(* IEC 61131-3 sources: SmartHomeNew/ (part 9) *)

(* ---- FB_System_Scenario_Arbitration.st ---- *)
// ==============================================================================
// System scenario arbitration helper
//
// Internal helper for PRG_System.
// Owns scenario request validation, priority resolution, fail-safe clamp,
// degraded-mode adaptation, policy logging, and FB_Scenario_Manager call.
// ==============================================================================
FUNCTION_BLOCK FB_System_Scenario_Arbitration
VAR_INPUT
    VI_System_Time_MS : UDINT;
    VI_IsActivePLC : BOOL;
    VI_System_Mode : E_System_Operating_Mode;
    VI_Security_Armed : BOOL;
END_VAR

VAR_IN_OUT
    VIO_Scenario_Req_Operator : E_SCENARIO_TYPE;
    VIO_Scenario_Req_Gateway : E_SCENARIO_TYPE;
    VIO_Scenario_Req_Rule : E_SCENARIO_TYPE;
    VIO_Scenario_Req_Final : E_SCENARIO_TYPE;
    VIO_Scenario_Intent : E_SCENARIO_TYPE;
    VIO_Scenario_Source : E_SCENARIO_SOURCE;
END_VAR

VAR
    fbLogEvent : FB_LogEvent;
    fbScenarioManager : FB_Scenario_Manager;
    L_Restore_Target : E_SCENARIO_TYPE;
END_VAR

// === SCENARIO REQUEST VALIDATION ===
// Normalize invalid values to NONE to avoid corrupt inputs.
// Actual enum range in E_SCENARIO_TYPE is 0..7.
IF TO_USINT(VIO_Scenario_Req_Operator) > 7 THEN
    VIO_Scenario_Req_Operator := E_SCENARIO_TYPE.SCENARIO_NONE;
END_IF;

IF TO_USINT(VIO_Scenario_Req_Gateway) > 7 THEN
    VIO_Scenario_Req_Gateway := E_SCENARIO_TYPE.SCENARIO_NONE;
END_IF;

IF TO_USINT(VIO_Scenario_Req_Rule) > 7 THEN
    VIO_Scenario_Req_Rule := E_SCENARIO_TYPE.SCENARIO_NONE;
END_IF;

// === SCENARIO PRIORITY RESOLUTION ===
// Produces VIO_Scenario_Req_Final (TRACE ONLY, not executed directly)
IF VI_System_Mode = E_System_Operating_Mode.MODE_SAFE_STOP THEN
    VIO_Scenario_Req_Final := 0;
    VIO_Scenario_Source := SRC_SAFETY;
ELSIF VIO_Scenario_Req_Operator <> 0 THEN
    VIO_Scenario_Req_Final := VIO_Scenario_Req_Operator;
    VIO_Scenario_Source := SRC_OPERATOR;
ELSIF VIO_Scenario_Req_Gateway <> 0 THEN
    VIO_Scenario_Req_Final := VIO_Scenario_Req_Gateway;
    VIO_Scenario_Source := SRC_GATEWAY;
ELSIF VIO_Scenario_Req_Rule <> 0 THEN
    VIO_Scenario_Req_Final := VIO_Scenario_Req_Rule;
    VIO_Scenario_Source := SRC_RULE;
ELSE
    VIO_Scenario_Req_Final := GVL_STATUS.G_Current_Scenario;
    VIO_Scenario_Source := SRC_NONE;
END_IF;

VIO_Scenario_Intent := VIO_Scenario_Req_Final;

// === FAIL-SAFE SCENARIO CLAMP ===
CASE VI_System_Mode OF
    E_System_Operating_Mode.MODE_SAFE_STOP:
        VIO_Scenario_Intent := E_SCENARIO_TYPE.SCENARIO_NONE;

    E_System_Operating_Mode.MODE_FREEZE_PROTECTION:
        VIO_Scenario_Intent := E_SCENARIO_TYPE.SCENARIO_NONE;

    E_System_Operating_Mode.MODE_DEGRADED:
        CASE VIO_Scenario_Intent OF
            E_SCENARIO_TYPE.SCENARIO_NONE,
            E_SCENARIO_TYPE.SCENARIO_PRESENCE,
            E_SCENARIO_TYPE.SCENARIO_AWAY,
            E_SCENARIO_TYPE.SCENARIO_SLEEP:
                ; // allowed in degraded
        ELSE
            VIO_Scenario_Intent := E_SCENARIO_TYPE.SCENARIO_NONE;
        END_CASE;
END_CASE;

// === CONTEXT FAIL-SAFE AUTOMATION ===
// If security is armed and no explicit source is requesting another scenario,
// force safe occupancy context to AWAY while system remains in MODE_NORMAL.
IF VI_System_Mode = E_System_Operating_Mode.MODE_NORMAL THEN
    IF VI_Security_Armed AND
       (VIO_Scenario_Req_Operator = E_SCENARIO_TYPE.SCENARIO_NONE) AND
       (VIO_Scenario_Req_Gateway = E_SCENARIO_TYPE.SCENARIO_NONE) AND
       (VIO_Scenario_Req_Rule = E_SCENARIO_TYPE.SCENARIO_NONE) AND
       (VIO_Scenario_Intent <> E_SCENARIO_TYPE.SCENARIO_AWAY) THEN

        IF (VIO_Scenario_Intent <> E_SCENARIO_TYPE.SCENARIO_NONE) AND
           (VIO_Scenario_Intent <> E_SCENARIO_TYPE.SCENARIO_AWAY) THEN
            GVL_POLICY.G_Away_Previous_Scenario := VIO_Scenario_Intent;
        ELSIF (GVL_STATUS.G_Current_Scenario <> E_SCENARIO_TYPE.SCENARIO_NONE) AND
              (GVL_STATUS.G_Current_Scenario <> E_SCENARIO_TYPE.SCENARIO_AWAY) THEN
            GVL_POLICY.G_Away_Previous_Scenario := GVL_STATUS.G_Current_Scenario;
        ELSE
            GVL_POLICY.G_Away_Previous_Scenario := E_SCENARIO_TYPE.SCENARIO_PRESENCE;
        END_IF;

        VIO_Scenario_Intent := E_SCENARIO_TYPE.SCENARIO_AWAY;
        VIO_Scenario_Source := SRC_POLICY;

        fbLogEvent(
            VI_Event_Type := 5,
            VI_Timestamp := VI_System_Time_MS,
            VI_Param1 := TO_UDINT(VIO_Scenario_Source),
            VI_Param2 := TO_UDINT(E_SCENARIO_TYPE.SCENARIO_AWAY)
        );
    END_IF;

    // When security is disarmed and no explicit source requests AWAY,
    // leave AWAY and return to the scenario captured before short-away arming.
    IF (NOT VI_Security_Armed) AND
       (VIO_Scenario_Req_Operator = E_SCENARIO_TYPE.SCENARIO_NONE) AND
       (VIO_Scenario_Req_Gateway = E_SCENARIO_TYPE.SCENARIO_NONE) AND
       (VIO_Scenario_Req_Rule = E_SCENARIO_TYPE.SCENARIO_NONE) AND
       (VIO_Scenario_Intent = E_SCENARIO_TYPE.SCENARIO_AWAY) AND
       GVL_POLICY.G_Away_Active THEN

        L_Restore_Target := GVL_POLICY.G_Away_Previous_Scenario;

        IF (L_Restore_Target = E_SCENARIO_TYPE.SCENARIO_NONE) OR
           (L_Restore_Target = E_SCENARIO_TYPE.SCENARIO_AWAY) THEN
            L_Restore_Target := E_SCENARIO_TYPE.SCENARIO_PRESENCE;
        END_IF;

        VIO_Scenario_Intent := L_Restore_Target;
        VIO_Scenario_Source := SRC_POLICY;
    END_IF;
END_IF;

// === DEGRADED-AWARE SCENARIO ADAPTATION ===
// Soft adaptation in degraded mode: keep explicit requests intact,
// but if no source is requesting a scenario, move behavior to a safer baseline.
IF VI_System_Mode = E_System_Operating_Mode.MODE_DEGRADED THEN
    IF (VIO_Scenario_Req_Operator = E_SCENARIO_TYPE.SCENARIO_NONE) AND
       (VIO_Scenario_Req_Gateway = E_SCENARIO_TYPE.SCENARIO_NONE) AND
       (VIO_Scenario_Req_Rule = E_SCENARIO_TYPE.SCENARIO_NONE) THEN

        IF VI_Security_Armed THEN
            IF VIO_Scenario_Intent <> E_SCENARIO_TYPE.SCENARIO_AWAY THEN
                IF (VIO_Scenario_Intent <> E_SCENARIO_TYPE.SCENARIO_NONE) AND
                   (VIO_Scenario_Intent <> E_SCENARIO_TYPE.SCENARIO_AWAY) THEN
                    GVL_POLICY.G_Away_Previous_Scenario := VIO_Scenario_Intent;
                ELSE
                    GVL_POLICY.G_Away_Previous_Scenario := E_SCENARIO_TYPE.SCENARIO_PRESENCE;
                END_IF;

                VIO_Scenario_Intent := E_SCENARIO_TYPE.SCENARIO_AWAY;
                VIO_Scenario_Source := SRC_POLICY;

                fbLogEvent(
                    VI_Event_Type := 6,
                    VI_Timestamp := VI_System_Time_MS,
                    VI_Param1 := TO_UDINT(VIO_Scenario_Source),
                    VI_Param2 := TO_UDINT(E_SCENARIO_TYPE.SCENARIO_AWAY)
                );
            END_IF;

        ELSIF VIO_Scenario_Intent = E_SCENARIO_TYPE.SCENARIO_PRESENCE THEN
            IF VIO_Scenario_Intent <> E_SCENARIO_TYPE.SCENARIO_SLEEP THEN
                VIO_Scenario_Intent := E_SCENARIO_TYPE.SCENARIO_SLEEP;
                VIO_Scenario_Source := SRC_POLICY;

                fbLogEvent(
                    VI_Event_Type := 7,
                    VI_Timestamp := VI_System_Time_MS,
                    VI_Param1 := TO_UDINT(VIO_Scenario_Source),
                    VI_Param2 := TO_UDINT(E_SCENARIO_TYPE.SCENARIO_SLEEP)
                );
            END_IF;
        END_IF;
    END_IF;
END_IF;

fbScenarioManager(
    VI_System_Time_MS := VI_System_Time_MS,
    VI_Activate_Request := VIO_Scenario_Intent,
    VI_IsActivePLC := VI_IsActivePLC,
    VI_System_Mode := VI_System_Mode,
    VO_Current_Scenario => GVL_STATUS.G_Current_Scenario
);

// >>> BULK_SYNC_ANCHOR: FB_System_Scenario_Arbitration <<<
END_FUNCTION_BLOCK

(* ---- FB_System_Timebase.st ---- *)
// ==============================================================================
// System timebase helper
//
// Internal helper for PRG_System.
// Owns PLC runtime clock projection into GVL_STATUS:
// - monotonic system milliseconds
// - time-of-day milliseconds
// - day of week / day of year rollover
// - TOD representation
// ==============================================================================
FUNCTION_BLOCK FB_System_Timebase
VAR
    L_Time_Diff : UDINT;
END_VAR

GVL_STATUS.G_System_Time_MS := TIME_TO_UDINT(TIME());

L_Time_Diff := SEL(
    GVL_STATUS.G_System_Time_MS >= GVL_STATUS.G_Last_System_Time_MS,
    GVL_STATUS.G_System_Time_MS - GVL_STATUS.G_Last_System_Time_MS,
    (4294967295 - GVL_STATUS.G_Last_System_Time_MS) + GVL_STATUS.G_System_Time_MS + 1
);

GVL_STATUS.G_Time_Of_Day_MS := (GVL_STATUS.G_Time_Of_Day_MS + L_Time_Diff) MOD 86400000;

IF GVL_STATUS.G_Time_Of_Day_MS < L_Time_Diff THEN
    GVL_STATUS.G_Current_Day := (GVL_STATUS.G_Current_Day MOD 7) + 1;
    GVL_STATUS.G_Day_Of_Year := (GVL_STATUS.G_Day_Of_Year MOD 365) + 1;
END_IF;

GVL_STATUS.G_Last_System_Time_MS := GVL_STATUS.G_System_Time_MS;
GVL_STATUS.G_Current_TOD := UDINT_TO_TOD(GVL_STATUS.G_Time_Of_Day_MS);

// >>> BULK_SYNC_ANCHOR: FB_System_Timebase <<<
END_FUNCTION_BLOCK

(* ---- FB_Time_Service.st ---- *)
FUNCTION_BLOCK FB_Time_Service
VAR
    L_Real_Now : UDINT;
    L_Elapsed : UDINT;
    L_Scaled_Delta : UDINT;
END_VAR

// read real time
L_Real_Now := GVL_STATUS.G_System_Time_MS;

// wrap-safe delta (real time base)
IF L_Real_Now >= GVL_TIME_SERVICE.G_Last_Now_MS THEN
    L_Elapsed := L_Real_Now - GVL_TIME_SERVICE.G_Last_Now_MS;
    GVL_TIME_SERVICE.G_Wrap_Detected := FALSE;
ELSE
    L_Elapsed := (16#FFFFFFFF - GVL_TIME_SERVICE.G_Last_Now_MS) + L_Real_Now + 1;
    GVL_TIME_SERVICE.G_Wrap_Detected := TRUE;
END_IF;

GVL_TIME_SERVICE.G_Last_Now_MS := L_Real_Now;

// --- SIMULATION MODE ---
IF GVL_TIME_SERVICE.G_Sim_Enabled THEN

    IF NOT GVL_TIME_SERVICE.G_Sim_Frozen THEN
        // scale delta
        L_Scaled_Delta := UDINT(REAL(L_Elapsed) * GVL_TIME_SERVICE.G_Sim_Time_Scale);

        // advance simulated absolute time
        GVL_TIME_SERVICE.G_Sim_Now_MS := GVL_TIME_SERVICE.G_Sim_Now_MS + L_Scaled_Delta;

        // advance TOD with wrap
        GVL_TIME_SERVICE.G_Sim_Time_Of_Day_MS := GVL_TIME_SERVICE.G_Sim_Time_Of_Day_MS + L_Scaled_Delta;

        IF GVL_TIME_SERVICE.G_Sim_Time_Of_Day_MS >= 86400000 THEN
            GVL_TIME_SERVICE.G_Sim_Time_Of_Day_MS := GVL_TIME_SERVICE.G_Sim_Time_Of_Day_MS MOD 86400000;
            GVL_TIME_SERVICE.G_Sim_Day_Of_Week := GVL_TIME_SERVICE.G_Sim_Day_Of_Week + 1;
            IF GVL_TIME_SERVICE.G_Sim_Day_Of_Week > 7 THEN
                GVL_TIME_SERVICE.G_Sim_Day_Of_Week := 1;
            END_IF;
        END_IF;
    END_IF;

    // publish simulated time
    GVL_TIME_SERVICE.G_Now_MS := GVL_TIME_SERVICE.G_Sim_Now_MS;
    GVL_TIME_SERVICE.G_Time_Of_Day_MS := GVL_TIME_SERVICE.G_Sim_Time_Of_Day_MS;
    GVL_TIME_SERVICE.G_Day_Of_Week := GVL_TIME_SERVICE.G_Sim_Day_Of_Week;

ELSE
    // publish real time
    GVL_TIME_SERVICE.G_Now_MS := L_Real_Now;
    GVL_TIME_SERVICE.G_Time_Of_Day_MS := GVL_STATUS.G_Time_Of_Day_MS;
    GVL_TIME_SERVICE.G_Day_Of_Week := INT(GVL_STATUS.G_Current_Day);
END_IF;

// publish delta (always based on real time)
GVL_TIME_SERVICE.G_Delta_MS := L_Elapsed;

END_FUNCTION_BLOCK

(* ---- FB_Trace_Logger.st ---- *)
FUNCTION_BLOCK FB_Trace_Logger
VAR_INPUT
    VI_Event_Code : INT;
    VI_System_Time : UDINT;
END_VAR

GVL_TRACE.G_Trace_Index := GVL_TRACE.G_Trace_Index + 1;
IF GVL_TRACE.G_Trace_Index > GVL_TRACE.G_Trace_Max THEN
    GVL_TRACE.G_Trace_Index := 1;
END_IF;

GVL_TRACE.G_Trace_Time[GVL_TRACE.G_Trace_Index] := VI_System_Time;
GVL_TRACE.G_Trace_Code[GVL_TRACE.G_Trace_Index] := VI_Event_Code;
END_FUNCTION_BLOCK

(* ---- FB_Trace_Write.st ---- *)
FUNCTION_BLOCK FB_Trace_Write
VAR_INPUT
    iLayer : E_Trace_Layer;
    iSource : E_Trace_Source;
    iReason : E_System_Reason_Code;
    iValueBool : BOOL;
    iValueReal : REAL;
    iText : STRING(120);
END_VAR

VAR
    L_Index : INT;
END_VAR

IF NOT GVL_TRACE.G_Trace_Enabled THEN RETURN; END_IF;

L_Index := GVL_TRACE.G_Trace_Write_Index;

GVL_TRACE.G_Trace_Buffer[L_Index].Timestamp_MS := GVL_TIME_SERVICE.G_Now_MS;
GVL_TRACE.G_Trace_Buffer[L_Index].Layer := iLayer;
GVL_TRACE.G_Trace_Buffer[L_Index].Source := iSource;
GVL_TRACE.G_Trace_Buffer[L_Index].Reason_Code := iReason;
GVL_TRACE.G_Trace_Buffer[L_Index].Value_Bool := iValueBool;
GVL_TRACE.G_Trace_Buffer[L_Index].Value_Real := iValueReal;
GVL_TRACE.G_Trace_Buffer[L_Index].Text := iText;

L_Index := L_Index + 1;
IF L_Index > 200 THEN L_Index := 1; END_IF;

GVL_TRACE.G_Trace_Write_Index := L_Index;

(* ---- FB_Trend_Analyzer.st ---- *)
FUNCTION_BLOCK FB_Trend_Analyzer
VAR_INPUT
    VI_Count      : INT;
END_VAR
VAR_IN_OUT
    VI_Data       : ARRAY[1..GVL_CONSTANTS.C_MAX_TREND_DATA_POINTS] OF REAL;
END_VAR
VAR_OUTPUT
    VO_Average    : REAL;
    VO_Max        : REAL;
    VO_Min        : REAL;
    VO_Trend_Up   : BOOL;
    VO_Trend_Down : BOOL;
END_VAR
VAR
    L_i   : INT;
    L_Sum : REAL;
END_VAR

VO_Average := 0.0;
VO_Max := 0.0;
VO_Min := 0.0;
VO_Trend_Up := FALSE;
VO_Trend_Down := FALSE;

IF VI_Count > 0 AND VI_Count <= GVL_CONSTANTS.C_MAX_TREND_DATA_POINTS THEN
    VO_Max := VI_Data[1];
    VO_Min := VI_Data[1];
    L_Sum := 0.0;

    FOR L_i := 1 TO VI_Count DO
        IF VI_Data[L_i] > VO_Max THEN VO_Max := VI_Data[L_i]; END_IF;
        IF VI_Data[L_i] < VO_Min THEN VO_Min := VI_Data[L_i]; END_IF;
        L_Sum := L_Sum + VI_Data[L_i];
    END_FOR;

    VO_Average := L_Sum / INT_TO_REAL(VI_Count);

    IF VI_Count >= 2 THEN
        VO_Trend_Up := (VI_Data[VI_Count] > VI_Data[1]);
        VO_Trend_Down := (VI_Data[VI_Count] < VI_Data[1]);
    END_IF;
END_IF;
END_FUNCTION_BLOCK

(* ---- FB_Trend_Logger.st ---- *)
FUNCTION_BLOCK FB_Trend_Logger
VAR_INPUT
    VI_System_Time_MS : UDINT;
    VI_Config : ST_Trend_Config;
    VI_Current_Value : REAL;
END_VAR
VAR_OUTPUT
    VO_Data : ST_Trend_Data;
END_VAR
VAR
    L_Last_Log_Time : UDINT;
    L_Last_Value : REAL;
    L_Deviation : REAL;
    L_Elapsed_Time : UDINT;
    L_Write_Index : UDINT;
END_VAR

IF NOT VI_Config.enabled THEN
    RETURN;
END_IF;

L_Deviation := ABS(VI_Current_Value - L_Last_Value);
L_Elapsed_Time := SEL(
    VI_System_Time_MS >= L_Last_Log_Time,
    VI_System_Time_MS - L_Last_Log_Time,
    (4294967295 - L_Last_Log_Time) + VI_System_Time_MS + 1
);

IF (L_Deviation >= (ABS(L_Last_Value) * VI_Config.deviation_threshold_percent / REAL#100.0)) OR
   (L_Elapsed_Time >= GVL_CONSTANTS.C_MS_IN_HOUR) THEN

    L_Write_Index := (VO_Data.record_count MOD 100) + 1;
    VO_Data.write_index := L_Write_Index;
    VO_Data.values[L_Write_Index] := VI_Current_Value;
    VO_Data.timestamps[L_Write_Index] := VI_System_Time_MS;
    VO_Data.record_count := VO_Data.record_count + 1;
    VO_Data.sum_values := VO_Data.sum_values + VI_Current_Value;
    VO_Data.config := VI_Config;

    L_Last_Value := VI_Current_Value;
    L_Last_Log_Time := VI_System_Time_MS;
END_IF;

END_FUNCTION_BLOCK

(* ---- FB_Valve_Test_Manager.st ---- *)
FUNCTION_BLOCK FB_Valve_Test_Manager
VAR_INPUT
    VI_System_Time_MS : UDINT;
    VI_IsActivePLC : BOOL;
END_VAR
VAR_IN_OUT
    VI_Valve_Currents : ARRAY[1..GVL_CONSTANTS.C_MAX_MANIFOLDS] OF REAL;
    VI_Valve_End_Switches : ARRAY[1..GVL_CONSTANTS.C_MAX_MANIFOLDS] OF BOOL;
    VI_Config : ARRAY[1..GVL_CONSTANTS.C_MAX_MANIFOLDS] OF ST_Valve_Test_Config;
END_VAR
VAR_OUTPUT
    VO_Test_Active : BOOL;
    VO_Current_Valve : INT; // Текущий тестируемый клапан
    VO_Valve_Cmd : ARRAY[1..GVL_CONSTANTS.C_MAX_MANIFOLDS] OF BOOL;
    VO_Test_Results : ARRAY[1..GVL_CONSTANTS.C_MAX_MANIFOLDS] OF BOOL; // TRUE = OK
    VO_Status_Msg : STRING(200);
END_VAR
VAR
    L_State : INT;
    L_Current_Valve : INT := 1;
    L_Test_Start_Time : UDINT;
    L_Last_Test_Time : ARRAY[1..GVL_CONSTANTS.C_MAX_MANIFOLDS] OF UDINT;
    L_i : INT;
    L_Need_Test : BOOL;
    L_Elapsed_Time : UDINT;
END_VAR

IF NOT VI_IsActivePLC THEN RETURN; END_IF;

CASE L_State OF
    0: // Ожидание
        VO_Test_Active := FALSE;
        L_Need_Test := FALSE;

        // Поиск клапана, которому нужен тест (раз в неделю)
        FOR L_i := 1 TO GVL_CONSTANTS.C_MAX_MANIFOLDS DO
            IF VI_Config[L_i].enabled AND ((VI_System_Time_MS - L_Last_Test_Time[L_i]) > (VI_Config[L_i].test_interval_days * 86400000)) THEN
                L_Current_Valve := L_i;
                L_Need_Test := TRUE;
                EXIT;
            END_IF;
        END_FOR;

        IF L_Need_Test THEN
            L_State := 1;
            L_Test_Start_Time := VI_System_Time_MS;
            VO_Test_Active := TRUE;
            VO_Current_Valve := L_Current_Valve;
            VO_Valve_Cmd[L_Current_Valve] := TRUE; // Открываем
            VO_Status_Msg := CONCAT('ТЕСТ КЛАПАНА ', INT_TO_STRING(L_Current_Valve));
            VO_Test_Results[L_Current_Valve] := TRUE; // Сброс результата
        END_IF;

    1: // Тестирование (ожидание открытия)
        L_Elapsed_Time := (VI_System_Time_MS - L_Test_Start_Time);

        IF VI_Valve_End_Switches[L_Current_Valve] THEN
            // Концевик сработал до истечения таймаута
            // Проверка тока
            IF ABS(VI_Valve_Currents[L_Current_Valve] - VI_Config[L_Current_Valve].Nominal_Current) > (VI_Config[L_Current_Valve].Nominal_Current * 0.2) THEN
                VO_Test_Results[L_Current_Valve] := FALSE; // Ошибка по току
            END_IF;

            GVL_Retain.G_Valve_Test_Results[L_Current_Valve] := VO_Test_Results[L_Current_Valve];

            VO_Valve_Cmd[L_Current_Valve] := FALSE; // Закрываем
            L_Test_Start_Time := VI_System_Time_MS; // Перезапускаем таймер для проверки закрытия
            L_State := 2;
        ELSIF L_Elapsed_Time > TO_UDINT(VI_Config[L_Current_Valve].nominal_close_time_sec * 1000.0) THEN
            // Таймаут открытия (заклинивание)
            VO_Test_Results[L_Current_Valve] := FALSE;
            GVL_Retain.G_Valve_Test_Results[L_Current_Valve] := FALSE;
            VO_Status_Msg := CONCAT('ОШИБКА: ЗАКЛИНИВАНИЕ КЛАПАНА ', INT_TO_STRING(L_Current_Valve));

            VO_Valve_Cmd[L_Current_Valve] := FALSE; // Закрываем
            L_Test_Start_Time := VI_System_Time_MS; // Перезапускаем таймер
            L_State := 2;
        END_IF;

    2: // Ожидание закрытия
        L_Elapsed_Time := (VI_System_Time_MS - L_Test_Start_Time);

        IF NOT VI_Valve_End_Switches[L_Current_Valve] THEN
            // Концевик разомкнулся (клапан закрыт)
            L_Last_Test_Time[L_Current_Valve] := VI_System_Time_MS;
            L_State := 0;
            IF VO_Test_Results[L_Current_Valve] THEN
                VO_Status_Msg := 'ТЕСТ ЗАВЕРШЕН УСПЕШНО';
            END_IF;
        ELSIF L_Elapsed_Time > TO_UDINT(VI_Config[L_Current_Valve].nominal_close_time_sec * 1000.0) THEN
            // Таймаут закрытия (заклинивание)
            VO_Test_Results[L_Current_Valve] := FALSE;
            GVL_Retain.G_Valve_Test_Results[L_Current_Valve] := FALSE;
            VO_Status_Msg := CONCAT('ОШИБКА: НЕ ЗАКРЫЛСЯ КЛАПАН ', INT_TO_STRING(L_Current_Valve));

            L_Last_Test_Time[L_Current_Valve] := VI_System_Time_MS;
            L_State := 0;
        END_IF;
ELSE
        // No fallback required
END_CASE;
END_FUNCTION_BLOCK

(* ---- FB_Vent_Output_Projection.st ---- *)
FUNCTION_BLOCK FB_Vent_Output_Projection
VAR_INPUT
    VI_Supply_Fans : ARRAY[1..GVL_CONSTANTS.C_MAX_SUPPLY_FANS] OF BYTE;
    VI_Exhaust_Fans : ARRAY[1..GVL_CONSTANTS.C_MAX_EXHAUST_FANS] OF BYTE;
END_VAR
VAR
    L_i : INT;
    L_Any_Fan_Active : BOOL;
END_VAR

// Convert ventilation manager BYTE outputs directly into IO-ready projection.
// PRG_Ventilation no longer needs to publish fan actuator values through GVL_STATE.

L_Any_Fan_Active := FALSE;

FOR L_i := 1 TO GVL_CONSTANTS.C_MAX_SUPPLY_FANS DO
    GVL_VENT_OUTPUT.AO_Supply_Fans[L_i] := BYTE_TO_UINT(VI_Supply_Fans[L_i]) * 10;
    IF VI_Supply_Fans[L_i] > 0 THEN
        L_Any_Fan_Active := TRUE;
    END_IF;
END_FOR;

FOR L_i := 1 TO GVL_CONSTANTS.C_MAX_EXHAUST_FANS DO
    GVL_VENT_OUTPUT.AO_Exhaust_Fans[L_i] := BYTE_TO_UINT(VI_Exhaust_Fans[L_i]) * 10;
    IF VI_Exhaust_Fans[L_i] > 0 THEN
        L_Any_Fan_Active := TRUE;
    END_IF;
END_FOR;

GVL_VENT_OUTPUT.DO_Vent_Enable := L_Any_Fan_Active;

END_FUNCTION_BLOCK
// >>> BULK_SYNC_ANCHOR: FB_Vent_Output_Projection <<<

(* ---- FB_Ventilation_System_Manager.st ---- *)
FUNCTION_BLOCK FB_Ventilation_System_Manager
VAR_INPUT
    VI_System_Time_MS : UDINT; // Системное время (мс)
    VI_IsActivePLC : BOOL; // Флаг: Данный ПЛК является ведущим
    VI_Outdoor_Temp : REAL; // Уличная температура воздуха (°C)
    VI_Current_Scenario : E_SCENARIO_TYPE; // Текущий глобальный сценарий
    VI_System_Mode : E_System_Operating_Mode; // Агрегированный режим работы системы
    VI_Config : ST_Ventilation_Global_Config; // Конфигурация системы вентиляции
    VI_Fire_Alarm : BOOL; // Сигнал пожарной тревоги
    VI_Gas_Alarm : BOOL; // Сигнал газовой тревоги
    VI_PV3_Boost_Req : BOOL; // Запрос форсирования ПВ-3 от газоанализатора (ТЗ 5.1)
    VI_Supply_100_Req : BOOL; // Запрос 100% притока (ТЗ 6.4)
    VI_Exhaust_100_Req : BOOL; // Запрос 100% вытяжки (ТЗ 6.4)
    VI_Supply_80_Req : BOOL; // Запрос 80% притока (ТЗ 5.4)
    VI_Vent_Stop : BOOL; // Запрос на остановку вентиляции (ТЗ 5.3)
    VI_IO_Modules_Online : ARRAY[1..GVL_CONSTANTS.C_MAX_MODULES] OF BOOL; // Статусы модулей ввода-вывода (только чтение)
END_VAR
VAR_IN_OUT
    VI_Supply_Temps : ARRAY[1..GVL_CONSTANTS.C_MAX_SUPPLY_TEMPS] OF REAL; // Температура приточного воздуха после калорифера
    VI_Room_Temps : ARRAY[1..16] OF REAL; // Температура в помещениях (°C)
    VI_Room_Humidities : ARRAY[1..16] OF REAL; // Влажность в помещениях (%)
    VI_Room_CO2 : ARRAY[1..16] OF REAL; // Уровень CO2 в помещениях (ppm)
    VI_Wet_Zone_Active : ARRAY[1..GVL_CONSTANTS.C_MAX_WET_ZONES] OF BOOL; // Сигналы включения света в санузлах (ТЗ 4.0)
    VI_Rule_Actions : ARRAY[1..GVL_CONSTANTS.C_MAX_RULES] OF ST_Rule_Action; // Действия от Rule Engine
END_VAR
VAR_OUTPUT
    VO_Supply_Fans : ARRAY[1..GVL_CONSTANTS.C_MAX_SUPPLY_FANS] OF BYTE; // Выход: Управление приточными вентиляторами (0-100%)
    VO_Exhaust_Fans : ARRAY[1..GVL_CONSTANTS.C_MAX_EXHAUST_FANS] OF BYTE; // Выход: Управление вытяжными вентиляторами (0-100%)
    VO_Heater_Power : ARRAY[1..GVL_CONSTANTS.C_MAX_BOILERS] OF REAL; // Выход: Мощность калориферов (0-100%)
    VO_Status_Msg : STRING(200); // Строковое сообщение о статусе
    VO_Ventilation_IO_Fault : BOOL; // Выход: диагностика потери связи с модулями ввода-вывода
    VO_Ventilation_Subsystem_Degraded : BOOL; // Выход: признак degraded-состояния подсистемы вентиляции
END_VAR
VAR
    L_Policy_Normal : BOOL;
    L_Policy_Safe_Stop : BOOL;
    L_Policy_Degraded : BOOL;
    L_Policy_Freeze_Protection : BOOL;
    L_i : INT;
    L_j : INT;
    L_Max_CO2 : REAL;
    L_Max_Hum : REAL;
    L_Base_Speed : BYTE;
    L_Target_Temp : REAL;
    L_PID_Heaters : ARRAY[1..GVL_CONSTANTS.C_MAX_BOILERS] OF FB_PID_Controller;
    L_Wet_Zone_Timers : ARRAY[1..GVL_CONSTANTS.C_MAX_WET_ZONES] OF FB_System_Timer_TOF; // Таймеры выбега для вытяжек санузлов
END_VAR

// Reset retained outputs on every call before any early return.
FOR L_i := 1 TO GVL_CONSTANTS.C_MAX_SUPPLY_FANS DO
    VO_Supply_Fans[L_i] := 0;
END_FOR;

FOR L_i := 1 TO GVL_CONSTANTS.C_MAX_EXHAUST_FANS DO
    VO_Exhaust_Fans[L_i] := 0;
END_FOR;

FOR L_i := 1 TO GVL_CONSTANTS.C_MAX_BOILERS DO
    VO_Heater_Power[L_i] := 0.0;
END_FOR;

VO_Status_Msg := '';
VO_Ventilation_IO_Fault := FALSE;
VO_Ventilation_Subsystem_Degraded := FALSE;

// ========================================
// Ventilation policy layer
// ========================================
L_Policy_Normal := (VI_System_Mode = E_System_Operating_Mode.MODE_NORMAL);
L_Policy_Safe_Stop := (VI_System_Mode = E_System_Operating_Mode.MODE_SAFE_STOP);
L_Policy_Degraded := (VI_System_Mode = E_System_Operating_Mode.MODE_DEGRADED);
L_Policy_Freeze_Protection := (VI_System_Mode = E_System_Operating_Mode.MODE_FREEZE_PROTECTION);

IF NOT VI_IsActivePLC THEN
    VO_Status_Msg := 'ВЕНТИЛЯЦИЯ: РЕЗЕРВНЫЙ ПЛК';
    RETURN;
END_IF;

// Проверка связи с модулями ввода-вывода
FOR L_i := 1 TO GVL_CONSTANTS.C_MAX_MODULES DO
    IF NOT VI_IO_Modules_Online[L_i] THEN
        VO_Ventilation_IO_Fault := TRUE;
        VO_Status_Msg := 'ОШИБКА: Потеря связи с модулями ввода-вывода';
        RETURN;
    END_IF;
END_FOR;

// =========================
// SYSTEM MODE / HARD REQUEST OVERRIDES
// =========================
IF L_Policy_Safe_Stop OR VI_Vent_Stop THEN
    IF VI_Vent_Stop THEN
        VO_Status_Msg := 'ВЕНТИЛЯЦИЯ: ОСТАНОВЛЕНА ПО КОМАНДЕ';
    ELSE
        VO_Status_Msg := 'ВЕНТИЛЯЦИЯ: ОСТАНОВЛЕНА POLICY SAFE_STOP';
    END_IF;
    RETURN;
END_IF;

IF L_Policy_Degraded THEN
    VO_Ventilation_Subsystem_Degraded := TRUE;
    VO_Status_Msg := 'ВЕНТИЛЯЦИЯ: DEGRADED POLICY';
END_IF;

IF L_Policy_Freeze_Protection THEN
    VO_Status_Msg := 'ВЕНТИЛЯЦИЯ: FREEZE_PROTECTION POLICY (stop)';
    RETURN;
END_IF;

// 1. Определение базовой скорости и целевой температуры по сценарию (ТЗ 7.1)
CASE VI_Current_Scenario OF
    E_SCENARIO_TYPE.SCENARIO_AWAY:
        L_Base_Speed := VI_Config.Scenario_Modes[3].Base_Fan_Speed;
        L_Target_Temp := VI_Config.Scenario_Modes[3].Target_Temp;
    E_SCENARIO_TYPE.SCENARIO_SLEEP:
        L_Base_Speed := VI_Config.Scenario_Modes[2].Base_Fan_Speed;
        L_Target_Temp := VI_Config.Scenario_Modes[2].Target_Temp;
    ELSE // PRESENCE, MORNING, EVENING
        L_Base_Speed := VI_Config.Scenario_Modes[1].Base_Fan_Speed;
        L_Target_Temp := VI_Config.Scenario_Modes[1].Target_Temp;
END_CASE;

// 2. Логика управления приточными установками (П-1, П-2, П-3)
IF NOT L_Policy_Degraded THEN
    FOR L_i := 1 TO GVL_CONSTANTS.C_MAX_SUPPLY_FANS DO
        IF L_i <= GVL_CONSTANTS.C_MAX_SUPPLY_TEMPS THEN
            L_PID_Heaters[L_i](
                VI_SetPoint := L_Target_Temp,
                VI_ProcessValue := VI_Supply_Temps[L_i],
                VI_Kp := 4.0, VI_Tn := 120.0, VI_Tv := 0.0,
                VI_Y_Min := 0.0, VI_Y_Max := 100.0, VI_Cycle_Time_S := 1.0,
                VO_Output => VO_Heater_Power[L_i]
            );
        END_IF;

        VO_Supply_Fans[L_i] := L_Base_Speed;

        FOR L_j := 1 TO GVL_CONSTANTS.C_MAX_RULES DO
            IF VI_Rule_Actions[L_j].Active AND VI_Rule_Actions[L_j].Target_ID = L_i THEN
                IF VI_Rule_Actions[L_j].Action_Type = E_Rule_Action_Type.ACTION_SET_VENTILATION THEN
                    VO_Supply_Fans[L_i] := REAL_TO_BYTE(VI_Rule_Actions[L_j].Value);
                END_IF;
            END_IF;
        END_FOR;
    END_FOR;
END_IF;

// 3. Логика управления вытяжными установками (В-1 .. В-5)
FOR L_i := 1 TO GVL_CONSTANTS.C_MAX_EXHAUST_FANS DO
    VO_Exhaust_Fans[L_i] := L_Base_Speed;

    FOR L_j := 1 TO GVL_CONSTANTS.C_MAX_WET_ZONES DO
        IF VI_Config.wet_zone_to_exhaust_map[L_j] = L_i THEN
            L_Wet_Zone_Timers[L_j](IN := VI_Wet_Zone_Active[L_j], PT := T#5m, VI_System_Time_MS := VI_System_Time_MS);
            IF VI_Wet_Zone_Active[L_j] THEN
                VO_Exhaust_Fans[L_i] := 80;
            ELSIF L_Wet_Zone_Timers[L_j].Q THEN
                VO_Exhaust_Fans[L_i] := 50;
            END_IF;
        END_IF;
    END_FOR;
END_FOR;

// ========================================
// OPERATIONAL REQUEST OVERRIDES
// ========================================
IF NOT L_Policy_Degraded THEN
    IF VI_Supply_100_Req THEN
        FOR L_i := 1 TO GVL_CONSTANTS.C_MAX_SUPPLY_FANS DO
            VO_Supply_Fans[L_i] := 100;
        END_FOR;
    ELSIF VI_Supply_80_Req THEN
        FOR L_i := 1 TO GVL_CONSTANTS.C_MAX_SUPPLY_FANS DO
            IF VO_Supply_Fans[L_i] < 80 THEN
                VO_Supply_Fans[L_i] := 80;
            END_IF;
        END_FOR;
    END_IF;

    IF VI_PV3_Boost_Req THEN
        IF GVL_CONSTANTS.C_MAX_SUPPLY_FANS >= 3 THEN
            VO_Supply_Fans[3] := 100;
        END_IF;
    END_IF;
END_IF;

IF VI_Exhaust_100_Req THEN
    FOR L_i := 1 TO GVL_CONSTANTS.C_MAX_EXHAUST_FANS DO
        VO_Exhaust_Fans[L_i] := 100;
    END_FOR;
END_IF;

// ========================================
// VENT_FINAL_CLAMP
// ========================================
IF L_Policy_Degraded THEN
    FOR L_i := 1 TO GVL_CONSTANTS.C_MAX_SUPPLY_FANS DO
        VO_Supply_Fans[L_i] := 0;
    END_FOR;
    FOR L_i := 1 TO GVL_CONSTANTS.C_MAX_BOILERS DO
        VO_Heater_Power[L_i] := 0.0;
    END_FOR;
    FOR L_i := 1 TO GVL_CONSTANTS.C_MAX_EXHAUST_FANS DO
        VO_Exhaust_Fans[L_i] := MIN(VO_Exhaust_Fans[L_i], VI_Config.Degraded_Exhaust_Limit);
    END_FOR;
END_IF;

// 4. Формирование статусного сообщения
IF L_Policy_Degraded THEN
    VO_Status_Msg := 'ВЕНТИЛЯЦИЯ: DEGRADED POLICY';
ELSIF VI_PV3_Boost_Req OR VI_Supply_100_Req OR VI_Exhaust_100_Req OR VI_Supply_80_Req THEN
    VO_Status_Msg := 'Вентиляция: активен операционный boost/request';
ELSE
    VO_Status_Msg := 'Вентиляция работает в штатном режиме';
END_IF;
// >>> BULK_SYNC_ANCHOR: FB_Ventilation_System_Manager <<<
END_FUNCTION_BLOCK

(* ---- FB_Watchdog.st ---- *)
FUNCTION_BLOCK FB_Watchdog
VAR_INPUT
    VI_System_Time_MS : UDINT;
    VI_Timeout_MS     : UDINT := 2000;
END_VAR

VAR_OUTPUT
    VO_Alive          : BOOL;
    VO_Watchdog_Fault : BOOL;
    VO_Cycle_DT_MS    : UDINT;
END_VAR

VAR
    L_Initialized    : BOOL := FALSE;
    L_Last_Call_MS   : UDINT := 0;
    L_DT_MS          : UDINT := 0;
END_VAR

IF NOT L_Initialized THEN
    L_Initialized := TRUE;
    L_Last_Call_MS := VI_System_Time_MS;
    VO_Cycle_DT_MS := 0;
    VO_Watchdog_Fault := FALSE;
    VO_Alive := TRUE;
    RETURN;
END_IF;

// Measure real time gap between successive calls
L_DT_MS := (SEL(VI_System_Time_MS >= L_Last_Call_MS, VI_System_Time_MS - L_Last_Call_MS, (4294967295 - L_Last_Call_MS) + VI_System_Time_MS + 1));
VO_Cycle_DT_MS := L_DT_MS;

// Fault if the task/cycle resumed after an abnormal pause
VO_Watchdog_Fault := (L_DT_MS > VI_Timeout_MS);
VO_Alive := NOT VO_Watchdog_Fault;

// Store current timestamp for next cycle
L_Last_Call_MS := VI_System_Time_MS;
// >>> BULK_SYNC_ANCHOR: FB_Watchdog <<<

(* ---- FB_Water_Hardware_Binding_Runtime.st ---- *)
FUNCTION_BLOCK FB_Water_Hardware_Binding_Runtime
VAR_INPUT
    VI_Enable : BOOL;
    VI_System_Time_MS : UDINT;
END_VAR
VAR
    L_i : INT;
    L_Binding : ST_IO_Binding_Record;
    L_Any_Invalid : BOOL;
    L_Any_Missing : BOOL;
END_VAR

IF NOT VI_Enable THEN
    GVL_IO_Binding_Runtime.G_Runtime_Valid := FALSE;
    RETURN;
END_IF;

FOR L_i := 1 TO GVL_CONSTANTS.C_MAX_FLOOD_SENSORS DO

    // Flood sensor binding validation.
    L_Binding :=
        GVL_IO_Binding_Config.G_Flood_Sensor_Binding[L_i];

    IF NOT L_Binding.Binding_Valid THEN
        L_Any_Missing := TRUE;
    END_IF;

    // Valve feedback binding validation.
    L_Binding :=
        GVL_IO_Binding_Config.G_Water_Valve_Close_FB_Binding[L_i];

    IF L_Binding.Required
       AND NOT L_Binding.Binding_Valid THEN

        L_Any_Invalid := TRUE;

    END_IF;

END_FOR;

GVL_IO_Binding_Runtime.G_Any_Invalid_Binding :=
    L_Any_Invalid;

GVL_IO_Binding_Runtime.G_Any_Missing_Binding :=
    L_Any_Missing;

GVL_IO_Binding_Runtime.G_Runtime_Valid := TRUE;
GVL_IO_Binding_Runtime.G_Last_Update_MS := VI_System_Time_MS;

IF L_Any_Invalid THEN
    GVL_IO_Binding_Runtime.G_Status_Code := 2;
    GVL_IO_Binding_Runtime.G_Status_Text :=
        'Hardware binding invalid';
ELSIF L_Any_Missing THEN
    GVL_IO_Binding_Runtime.G_Status_Code := 1;
    GVL_IO_Binding_Runtime.G_Status_Text :=
        'Hardware binding incomplete';
ELSE
    GVL_IO_Binding_Runtime.G_Status_Code := 0;
    GVL_IO_Binding_Runtime.G_Status_Text :=
        'Hardware binding runtime healthy';
END_IF;

END_FUNCTION_BLOCK

(* ---- FB_Water_Hydraulic_Topology_Validator.st ---- *)
FUNCTION_BLOCK FB_Water_Hydraulic_Topology_Validator
VAR_INPUT
    VI_Enable : BOOL;
    VI_System_Time_MS : UDINT;
END_VAR
VAR
    L_i : INT;

    L_Node : ST_Water_Hydraulic_Topology_Node;
    L_Group : ST_Water_Hydraulic_Isolation_Group;
    L_Validation : ST_Water_Topology_Validation_State;

    L_Empty_Node : ST_Water_Hydraulic_Topology_Node;
    L_Empty_Group : ST_Water_Hydraulic_Isolation_Group;
    L_Empty_Validation : ST_Water_Topology_Validation_State;

    L_Any_Invalid : BOOL;
    L_Any_Ambiguous : BOOL;
    L_Any_Fallback : BOOL;
END_VAR

IF NOT VI_Enable THEN
    GVL_Water_Topology_Validation.G_Runtime_Valid := FALSE;
    RETURN;
END_IF;

L_Any_Invalid := FALSE;
L_Any_Ambiguous := FALSE;
L_Any_Fallback := FALSE;

FOR L_i := 1 TO GVL_CONSTANTS.C_MAX_FLOOD_SENSORS DO

    L_Node := L_Empty_Node;
    L_Node.Runtime_Valid := TRUE;

    L_Node.Sensor_Id := TO_UINT(L_i);
    L_Node.Hydraulic_Zone_Id :=
        GVL_Water_Runtime_Projection.G_Leak_Runtime_State[L_i].Hydraulic_Zone_Id;

    L_Node.Valve_Group_Id :=
        GVL_Water_Runtime_Projection.G_Leak_Runtime_State[L_i].Valve_Group_Id;

    L_Node.Isolation_Group_Id :=
        L_Node.Valve_Group_Id;

    L_Node.Hydraulic_Segment_Id :=
        L_Node.Hydraulic_Zone_Id;

    L_Node.Fallback_Domain_Id := 1;

    // Validation.
    L_Node.Mapping_Valid :=
        L_Node.Valve_Group_Id <> 0;

    IF NOT L_Node.Mapping_Valid THEN
        L_Node.Global_Fallback_Required := TRUE;
        L_Node.Status_Code := 1;
        L_Node.Status_Text := 'Missing valve group';
    ELSE
        L_Node.Selective_Isolation_Allowed := TRUE;
        L_Node.Status_Code := 0;
        L_Node.Status_Text := 'Topology valid';
    END_IF;

    // Shared valve-group detection.
    IF L_Node.Valve_Group_Id = 3 THEN
        L_Node.Shared_Valve_Group := TRUE;
    END_IF;

    // Isolation group publication.
    L_Group := L_Empty_Group;
    L_Group.Runtime_Valid := TRUE;

    L_Group.Isolation_Group_Id :=
        L_Node.Isolation_Group_Id;

    L_Group.Valve_Group_Id :=
        L_Node.Valve_Group_Id;

    L_Group.Fallback_Domain_Id :=
        L_Node.Fallback_Domain_Id;

    L_Group.Shared_Sensor_Count :=
        SEL(L_Node.Shared_Valve_Group, 1, 2);

    L_Group.Isolation_Valid :=
        L_Node.Mapping_Valid;

    L_Group.Isolation_Ambiguous :=
        L_Node.Mapping_Ambiguous;

    L_Group.Selective_Isolation_Allowed :=
        L_Node.Selective_Isolation_Allowed;

    L_Group.Global_Fallback_Required :=
        L_Node.Global_Fallback_Required;

    // Validation publication.
    L_Validation := L_Empty_Validation;
    L_Validation.Runtime_Valid := TRUE;

    L_Validation.Runtime_System_Time_MS :=
        VI_System_Time_MS;

    L_Validation.Sensor_Id :=
        L_Node.Sensor_Id;

    L_Validation.Topology_Valid :=
        L_Node.Mapping_Valid;

    L_Validation.Topology_Ambiguous :=
        L_Node.Mapping_Ambiguous;

    L_Validation.Isolation_Path_Valid :=
        L_Group.Isolation_Valid;

    L_Validation.Shared_Valve_Group :=
        L_Node.Shared_Valve_Group;

    L_Validation.Missing_Valve_Group :=
        NOT L_Node.Mapping_Valid;

    L_Validation.Selective_Isolation_Allowed :=
        L_Node.Selective_Isolation_Allowed;

    L_Validation.Global_Fallback_Required :=
        L_Node.Global_Fallback_Required;

    IF L_Validation.Global_Fallback_Required THEN
        L_Validation.Status_Code := 1;
        L_Validation.Status_Text :=
            'Global fallback required';
    ELSE
        L_Validation.Status_Code := 0;
        L_Validation.Status_Text :=
            'Topology validation healthy';
    END_IF;

    GVL_Water_Hydraulic_Topology.G_Topology_Node[L_i] :=
        L_Node;

    GVL_Water_Hydraulic_Topology.G_Isolation_Group[L_i] :=
        L_Group;

    GVL_Water_Topology_Validation.G_Validation_State[L_i] :=
        L_Validation;

    L_Any_Invalid :=
        L_Any_Invalid
        OR NOT L_Validation.Topology_Valid;

    L_Any_Ambiguous :=
        L_Any_Ambiguous
        OR L_Validation.Topology_Ambiguous;

    L_Any_Fallback :=
        L_Any_Fallback
        OR L_Validation.Global_Fallback_Required;

END_FOR;

GVL_Water_Hydraulic_Topology.G_Any_Ambiguous :=
    L_Any_Ambiguous;

GVL_Water_Hydraulic_Topology.G_Any_Global_Fallback_Required :=
    L_Any_Fallback;

GVL_Water_Hydraulic_Topology.G_Runtime_Valid := TRUE;
GVL_Water_Hydraulic_Topology.G_Last_Update_MS := VI_System_Time_MS;

GVL_Water_Topology_Validation.G_Any_Invalid :=
    L_Any_Invalid;

GVL_Water_Topology_Validation.G_Any_Ambiguous :=
    L_Any_Ambiguous;

GVL_Water_Topology_Validation.G_Any_Global_Fallback_Required :=
    L_Any_Fallback;

GVL_Water_Topology_Validation.G_Runtime_Valid := TRUE;
GVL_Water_Topology_Validation.G_Last_Update_MS := VI_System_Time_MS;

END_FUNCTION_BLOCK

(* ---- FB_Water_Isolation_Authority_Arbitrator.st ---- *)
FUNCTION_BLOCK FB_Water_Isolation_Authority_Arbitrator
VAR_INPUT
    VI_Enable : BOOL;
    VI_System_Time_MS : UDINT;
END_VAR
VAR
    L_i : INT;
    L_Group : INT;
    L_Runtime : ST_Water_Isolation_Runtime_State;
    L_Traversal : ST_Water_Graph_Traversal_State;
    L_Authority : ST_Water_Isolation_Authority_State;
    L_Empty_Authority : ST_Water_Isolation_Authority_State;
    L_Any_Selective : BOOL;
    L_Any_Global : BOOL;
    L_Any_Denied : BOOL;
    L_Active_Group_Count : INT;
    L_Group_Active : ARRAY[1..GVL_CONSTANTS.C_MAX_FLOOD_VALVES] OF BOOL;
    L_Multiple_Groups_Active : BOOL;
END_VAR

IF NOT VI_Enable THEN
    GVL_Water_Isolation_Authority.G_Authority_Valid := FALSE;
    RETURN;
END_IF;

L_Any_Selective := FALSE;
L_Any_Global := FALSE;
L_Any_Denied := FALSE;
L_Active_Group_Count := 0;

FOR L_i := 1 TO GVL_CONSTANTS.C_MAX_FLOOD_VALVES DO
    L_Group_Active[L_i] := FALSE;
END_FOR;

// Count distinct logical leak zones/groups, not raw sensor count. Multiple
// sensors in the same zone must keep selective authority for that zone.
FOR L_i := 1 TO GVL_CONSTANTS.C_MAX_FLOOD_SENSORS DO
    L_Runtime := GVL_Water_Isolation_Runtime.G_Isolation_Runtime_State[L_i];

    IF L_Runtime.Isolation_Requested THEN
        L_Group := UINT_TO_INT(L_Runtime.Valve_Group_Id);

        IF (L_Group >= 1) AND (L_Group <= GVL_CONSTANTS.C_MAX_FLOOD_VALVES) THEN
            L_Group_Active[L_Group] := TRUE;
        ELSE
            L_Any_Global := TRUE;
        END_IF;
    END_IF;
END_FOR;

FOR L_i := 1 TO GVL_CONSTANTS.C_MAX_FLOOD_VALVES DO
    IF L_Group_Active[L_i] THEN
        L_Active_Group_Count := L_Active_Group_Count + 1;
    END_IF;
END_FOR;

L_Multiple_Groups_Active := L_Active_Group_Count > 1;

FOR L_i := 1 TO GVL_CONSTANTS.C_MAX_FLOOD_SENSORS DO

    L_Runtime := GVL_Water_Isolation_Runtime.G_Isolation_Runtime_State[L_i];
    L_Traversal := GVL_Water_Orchestration.G_Traversal_State[L_i];

    L_Authority := L_Empty_Authority;
    L_Authority.Decision_Valid := TRUE;
    L_Authority.Decision_System_Time_MS := VI_System_Time_MS;

    L_Authority.Isolation_Requested := L_Runtime.Isolation_Requested;
    L_Authority.Selective_Candidate := L_Runtime.Selective_Isolation_Requested;
    L_Authority.Global_Fallback_Candidate := L_Runtime.Global_Isolation_Requested;

    L_Authority.Hydraulic_Zone_Id := L_Runtime.Hydraulic_Zone_Id;
    L_Authority.Isolation_Group_Id := L_Runtime.Isolation_Group_Id;
    L_Authority.Valve_Group_Id := L_Runtime.Valve_Group_Id;

    // Orchestration-derived authority.
    L_Authority.Mapping_Valid := L_Traversal.Traversal_Valid;

    L_Authority.Deterministic_Target_Valid :=
        (L_Runtime.Valve_Group_Id <> 0)
        AND NOT L_Traversal.Traversal_Conflict
        AND NOT L_Traversal.Traversal_Ambiguous;

    L_Authority.Safety_Context_Allows_Selective :=
        NOT GVL_INTENT_SAFETY.I_Water_Main_Close_Required;

    IF NOT L_Authority.Isolation_Requested THEN

        L_Authority.Decision_Code := 0;
        L_Authority.Decision_Text := 'No authority required';

    ELSIF L_Multiple_Groups_Active THEN

        L_Authority.Global_Fallback_Required := TRUE;
        L_Authority.Authority_Denied := TRUE;

        L_Authority.Decision_Code := 3;
        L_Authority.Decision_Text := 'Global fallback authority active: multiple leak zones';

    ELSIF NOT L_Authority.Mapping_Valid
       OR NOT L_Authority.Deterministic_Target_Valid
       OR NOT L_Authority.Safety_Context_Allows_Selective THEN

        L_Authority.Global_Fallback_Required := TRUE;
        L_Authority.Authority_Denied := TRUE;

        L_Authority.Decision_Code := 2;
        L_Authority.Decision_Text := 'Global fallback authority active';

    ELSE

        L_Authority.Selective_Authority_Allowed := TRUE;

        L_Authority.Decision_Code := 10;
        L_Authority.Decision_Text := 'Selective authority granted';

    END_IF;

    GVL_Water_Isolation_Authority.G_Authority_State[L_i] :=
        L_Authority;

    L_Any_Selective :=
        L_Any_Selective
        OR L_Authority.Selective_Authority_Allowed;

    L_Any_Global :=
        L_Any_Global
        OR L_Authority.Global_Fallback_Required;

    L_Any_Denied :=
        L_Any_Denied
        OR L_Authority.Authority_Denied;

END_FOR;

GVL_Water_Isolation_Authority.G_Any_Selective_Authority_Allowed :=
    L_Any_Selective;

GVL_Water_Isolation_Authority.G_Any_Global_Fallback_Required :=
    L_Any_Global;

GVL_Water_Isolation_Authority.G_Any_Authority_Denied :=
    L_Any_Denied;

GVL_Water_Isolation_Authority.G_Authority_Valid := TRUE;
GVL_Water_Isolation_Authority.G_Last_Update_MS := VI_System_Time_MS;

IF L_Multiple_Groups_Active THEN
    GVL_Water_Isolation_Authority.G_Status_Code := 3;
    GVL_Water_Isolation_Authority.G_Status_Text :=
        'Global fallback authority active: multiple leak zones';
ELSIF L_Any_Global THEN
    GVL_Water_Isolation_Authority.G_Status_Code := 2;
    GVL_Water_Isolation_Authority.G_Status_Text :=
        'Global fallback authority active';
ELSIF L_Any_Selective THEN
    GVL_Water_Isolation_Authority.G_Status_Code := 1;
    GVL_Water_Isolation_Authority.G_Status_Text :=
        'Selective orchestration authority active';
ELSE
    GVL_Water_Isolation_Authority.G_Status_Code := 0;
    GVL_Water_Isolation_Authority.G_Status_Text :=
        'Authority arbitration healthy';
END_IF;

END_FUNCTION_BLOCK

(* ---- FB_Water_Isolation_Intent_Builder.st ---- *)
FUNCTION_BLOCK FB_Water_Isolation_Intent_Builder
VAR_INPUT
    VI_Enable : BOOL;
END_VAR
VAR
    L_i : INT;
    L_Group : INT;
    L_State : ST_Water_Isolation_Runtime_State;
    L_Any_Selective : BOOL;
    L_Global_Fallback : BOOL;
END_VAR

IF NOT VI_Enable THEN
    GVL_Water_Isolation_Intent.G_Intent_Valid := FALSE;
    RETURN;
END_IF;

L_Any_Selective := FALSE;
L_Global_Fallback := FALSE;

FOR L_i := 1 TO GVL_CONSTANTS.C_MAX_FLOOD_SENSORS DO
    GVL_Water_Isolation_Intent.G_Zone_Close_Requested[L_i] := FALSE;
END_FOR;

FOR L_i := 1 TO GVL_CONSTANTS.C_MAX_FLOOD_VALVES DO
    GVL_Water_Isolation_Intent.G_Valve_Group_Close_Requested[L_i] := FALSE;
END_FOR;

FOR L_i := 1 TO GVL_CONSTANTS.C_MAX_FLOOD_SENSORS DO

    L_State := GVL_Water_Isolation_Runtime.G_Isolation_Runtime_State[L_i];

    IF L_State.Selective_Isolation_Requested THEN

        IF (L_State.Hydraulic_Zone_Id >= 1)
           AND (L_State.Hydraulic_Zone_Id <= GVL_CONSTANTS.C_MAX_FLOOD_SENSORS) THEN

            GVL_Water_Isolation_Intent.G_Zone_Close_Requested[
                L_State.Hydraulic_Zone_Id
            ] := TRUE;

        END_IF;

        L_Group := UINT_TO_INT(L_State.Valve_Group_Id);

        IF (L_Group >= 1)
           AND (L_Group <= GVL_CONSTANTS.C_MAX_FLOOD_VALVES) THEN

            GVL_Water_Isolation_Intent.G_Valve_Group_Close_Requested[
                L_Group
            ] := TRUE;

        ELSE
            L_Global_Fallback := TRUE;
        END_IF;

        L_Any_Selective := TRUE;

    END_IF;

    IF L_State.Global_Isolation_Requested THEN
        L_Global_Fallback := TRUE;
    END_IF;

END_FOR;

GVL_Water_Isolation_Intent.G_Global_Isolation_Requested :=
    L_Global_Fallback;

GVL_Water_Isolation_Intent.G_Intent_Valid := TRUE;

IF L_Global_Fallback THEN
    GVL_Water_Isolation_Intent.G_Status_Code := 2;
    GVL_Water_Isolation_Intent.G_Status_Text :=
        'Global isolation fallback requested';
ELSIF L_Any_Selective THEN
    GVL_Water_Isolation_Intent.G_Status_Code := 1;
    GVL_Water_Isolation_Intent.G_Status_Text :=
        'Localized isolation intent available';
ELSE
    GVL_Water_Isolation_Intent.G_Status_Code := 0;
    GVL_Water_Isolation_Intent.G_Status_Text :=
        'No isolation intent active';
END_IF;

END_FUNCTION_BLOCK

(* ---- FB_Water_Isolation_Path_Resolver.st ---- *)
FUNCTION_BLOCK FB_Water_Isolation_Path_Resolver
VAR_INPUT
    VI_Enable : BOOL;
    VI_System_Time_MS : UDINT;
END_VAR
VAR
    L_i : INT;

    L_Edge : ST_Water_Hydraulic_Topology_Edge;
    L_Path : ST_Water_Isolation_Path_Runtime_State;
    L_Validation : ST_Water_Topology_Validation_State;

    L_Any_Shared_Trunk : BOOL;
    L_Any_Conflict : BOOL;
    L_Any_Fallback : BOOL;
END_VAR

IF NOT VI_Enable THEN
    GVL_Water_Hydraulic_Graph.G_Runtime_Valid := FALSE;
    RETURN;
END_IF;

FOR L_i := 1 TO GVL_CONSTANTS.C_MAX_FLOOD_SENSORS DO

    L_Validation :=
        GVL_Water_Topology_Validation.G_Validation_State[L_i];

    // Graph edge publication.
    L_Edge.Runtime_Valid := TRUE;

    L_Edge.Edge_Id := TO_UINT(L_i);

    L_Edge.Upstream_Segment_Id :=
        GVL_Water_Hydraulic_Topology.G_Topology_Node[L_i].Hydraulic_Segment_Id;

    L_Edge.Downstream_Segment_Id :=
        GVL_Water_Hydraulic_Topology.G_Topology_Node[L_i].Hydraulic_Zone_Id;

    L_Edge.Isolation_Group_Id :=
        GVL_Water_Hydraulic_Topology.G_Topology_Node[L_i].Isolation_Group_Id;

    L_Edge.Valve_Group_Id :=
        GVL_Water_Hydraulic_Topology.G_Topology_Node[L_i].Valve_Group_Id;

    // Shared trunk semantics.
    IF L_Edge.Valve_Group_Id = 3 THEN
        L_Edge.Shared_Trunk := TRUE;
        L_Edge.Cross_Zone_Dependency := TRUE;
    END_IF;

    L_Edge.Dependency_Valid :=
        L_Validation.Topology_Valid;

    L_Edge.Dependency_Ambiguous :=
        L_Validation.Topology_Ambiguous;

    L_Edge.Selective_Isolation_Allowed :=
        L_Validation.Selective_Isolation_Allowed;

    L_Edge.Global_Fallback_Required :=
        L_Validation.Global_Fallback_Required;

    // Isolation path runtime.
    L_Path.Runtime_Valid := TRUE;

    L_Path.Runtime_System_Time_MS :=
        VI_System_Time_MS;

    L_Path.Sensor_Id := TO_UINT(L_i);

    L_Path.Isolation_Path_Valid :=
        L_Edge.Dependency_Valid;

    L_Path.Isolation_Path_Ambiguous :=
        L_Edge.Dependency_Ambiguous;

    L_Path.Active_Isolation_Group_Id :=
        L_Edge.Isolation_Group_Id;

    L_Path.Active_Valve_Group_Id :=
        L_Edge.Valve_Group_Id;

    L_Path.Shared_Trunk_Impact :=
        L_Edge.Shared_Trunk;

    L_Path.Cross_Zone_Impact :=
        L_Edge.Cross_Zone_Dependency;

    L_Path.Selective_Isolation_Allowed :=
        L_Edge.Selective_Isolation_Allowed;

    L_Path.Global_Fallback_Required :=
        L_Edge.Global_Fallback_Required;

    // Multi-valve/shared-trunk path.
    IF L_Path.Shared_Trunk_Impact THEN
        L_Path.Multi_Valve_Path := TRUE;
    END_IF;

    // Conflict detection.
    IF L_Path.Isolation_Path_Ambiguous THEN
        L_Path.Conflict_Detected := TRUE;
    END_IF;

    // Conservative escalation.
    IF L_Path.Conflict_Detected THEN
        L_Path.Global_Fallback_Required := TRUE;
        L_Path.Selective_Isolation_Allowed := FALSE;

        L_Path.Status_Code := 2;
        L_Path.Status_Text :=
            'Isolation path conflict detected';

    ELSIF L_Path.Shared_Trunk_Impact THEN
        L_Path.Status_Code := 1;
        L_Path.Status_Text :=
            'Shared trunk isolation path active';

    ELSE
        L_Path.Status_Code := 0;
        L_Path.Status_Text :=
            'Isolation path resolved';
    END_IF;

    GVL_Water_Hydraulic_Graph.G_Topology_Edge[L_i] :=
        L_Edge;

    GVL_Water_Hydraulic_Graph.G_Isolation_Path[L_i] :=
        L_Path;

    L_Any_Shared_Trunk :=
        L_Any_Shared_Trunk
        OR L_Path.Shared_Trunk_Impact;

    L_Any_Conflict :=
        L_Any_Conflict
        OR L_Path.Conflict_Detected;

    L_Any_Fallback :=
        L_Any_Fallback
        OR L_Path.Global_Fallback_Required;

END_FOR;

GVL_Water_Hydraulic_Graph.G_Any_Shared_Trunk :=
    L_Any_Shared_Trunk;

GVL_Water_Hydraulic_Graph.G_Any_Conflict :=
    L_Any_Conflict;

GVL_Water_Hydraulic_Graph.G_Any_Global_Fallback_Required :=
    L_Any_Fallback;

GVL_Water_Hydraulic_Graph.G_Runtime_Valid := TRUE;
GVL_Water_Hydraulic_Graph.G_Last_Update_MS := VI_System_Time_MS;

IF L_Any_Conflict THEN
    GVL_Water_Hydraulic_Graph.G_Status_Code := 2;
    GVL_Water_Hydraulic_Graph.G_Status_Text :=
        'Hydraulic graph conflicts detected';
ELSIF L_Any_Shared_Trunk THEN
    GVL_Water_Hydraulic_Graph.G_Status_Code := 1;
    GVL_Water_Hydraulic_Graph.G_Status_Text :=
        'Shared trunk governance active';
ELSE
    GVL_Water_Hydraulic_Graph.G_Status_Code := 0;
    GVL_Water_Hydraulic_Graph.G_Status_Text :=
        'Hydraulic graph runtime healthy';
END_IF;

END_FUNCTION_BLOCK

(* ---- FB_Water_Isolation_Runtime_Projection.st ---- *)
FUNCTION_BLOCK FB_Water_Isolation_Runtime_Projection
VAR_INPUT
    VI_Enable : BOOL;
    VI_System_Time_MS : UDINT;
END_VAR
VAR
    L_i : INT;
    L_Leak_State : ST_Water_Leak_Runtime_State;
    L_Isolation_State : ST_Water_Isolation_Runtime_State;
    L_Traversal : ST_Water_Graph_Traversal_State;
    L_Empty_Isolation_State : ST_Water_Isolation_Runtime_State;
    L_Any_Isolation : BOOL;
    L_Any_Selective : BOOL;
    L_Global_Fallback : BOOL;
END_VAR

IF NOT VI_Enable THEN
    GVL_Water_Isolation_Runtime.G_Runtime_Valid := FALSE;
    RETURN;
END_IF;

L_Any_Isolation := FALSE;
L_Any_Selective := FALSE;
L_Global_Fallback := FALSE;

FOR L_i := 1 TO GVL_CONSTANTS.C_MAX_FLOOD_SENSORS DO

    L_Leak_State := GVL_Water_Runtime_Projection.G_Leak_Runtime_State[L_i];
    L_Traversal := GVL_Water_Orchestration.G_Traversal_State[L_i];

    L_Isolation_State := L_Empty_Isolation_State;
    L_Isolation_State.Projection_Valid := TRUE;
    L_Isolation_State.Projection_System_Time_MS := VI_System_Time_MS;

    L_Isolation_State.Hydraulic_Zone_Id := L_Leak_State.Hydraulic_Zone_Id;
    L_Isolation_State.Isolation_Group_Id := L_Leak_State.Isolation_Group_Id;
    L_Isolation_State.Valve_Group_Id := L_Traversal.Target_Valve_Group_Id;

    L_Isolation_State.Active_Global_Close_Path :=
        L_Leak_State.Active_Global_Close_Path;

    L_Isolation_State.Active_Safety_Latch :=
        L_Leak_State.Active_Safety_Leak_Latched;

    L_Isolation_State.Mapping_Valid :=
        L_Traversal.Traversal_Valid;

    L_Isolation_State.Fallback_To_Global_Required :=
        L_Traversal.Global_Fallback_Required;

    IF L_Leak_State.Leak_Confirmed THEN

        L_Isolation_State.Isolation_Requested := TRUE;

        IF L_Traversal.Selective_Path_Allowed
           AND NOT L_Traversal.Global_Fallback_Required THEN

            L_Isolation_State.Selective_Isolation_Requested := TRUE;
            L_Isolation_State.Reason_Code := 1;
            L_Isolation_State.Reason_Text :=
                'Selective orchestration path available';

        ELSE

            L_Isolation_State.Global_Isolation_Requested := TRUE;
            L_Isolation_State.Reason_Code := 2;
            L_Isolation_State.Reason_Text :=
                'Global fallback required';

        END_IF;

    END_IF;

    GVL_Water_Isolation_Runtime.G_Isolation_Runtime_State[L_i] :=
        L_Isolation_State;

    L_Any_Isolation :=
        L_Any_Isolation
        OR L_Isolation_State.Isolation_Requested;

    L_Any_Selective :=
        L_Any_Selective
        OR L_Isolation_State.Selective_Isolation_Requested;

    L_Global_Fallback :=
        L_Global_Fallback
        OR L_Isolation_State.Global_Isolation_Requested;

END_FOR;

GVL_Water_Isolation_Runtime.G_Any_Isolation_Requested :=
    L_Any_Isolation;

GVL_Water_Isolation_Runtime.G_Any_Selective_Isolation :=
    L_Any_Selective;

GVL_Water_Isolation_Runtime.G_Global_Fallback_Required :=
    L_Global_Fallback;

GVL_Water_Isolation_Runtime.G_Runtime_Valid := TRUE;
GVL_Water_Isolation_Runtime.G_Last_Update_MS := VI_System_Time_MS;

IF L_Global_Fallback THEN
    GVL_Water_Isolation_Runtime.G_Status_Code := 2;
    GVL_Water_Isolation_Runtime.G_Status_Text :=
        'Global isolation fallback required';
ELSIF L_Any_Selective THEN
    GVL_Water_Isolation_Runtime.G_Status_Code := 1;
    GVL_Water_Isolation_Runtime.G_Status_Text :=
        'Selective orchestration active';
ELSE
    GVL_Water_Isolation_Runtime.G_Status_Code := 0;
    GVL_Water_Isolation_Runtime.G_Status_Text :=
        'Isolation runtime active';
END_IF;

END_FUNCTION_BLOCK

(* ---- FB_Water_Leak_Runtime_Projection.st ---- *)
FUNCTION_BLOCK FB_Water_Leak_Runtime_Projection
VAR_INPUT
    VI_Enable : BOOL;
    VI_System_Time_MS : UDINT;
END_VAR
VAR
    L_i : INT;
    L_Group : INT;
    L_Runtime_State : ST_Water_Leak_Runtime_State;
    L_Global_Leak : BOOL;
    L_Global_Warning : BOOL;
END_VAR

IF NOT VI_Enable THEN
    GVL_Water_Runtime_Projection.G_Projection_Valid := FALSE;
    RETURN;
END_IF;

L_Global_Leak := FALSE;
L_Global_Warning := FALSE;

FOR L_i := 1 TO GVL_CONSTANTS.C_MAX_FLOOD_SENSORS DO

    L_Runtime_State.Projection_Valid := FALSE;
    L_Runtime_State.Projection_Valid := TRUE;
    L_Runtime_State.Projection_System_Time_MS := VI_System_Time_MS;
    L_Runtime_State.Physical_Sensor_Index := TO_UINT(L_i);
    L_Runtime_State.Physical_Input_Valid := TRUE;
    L_Runtime_State.Leak_Warning_Active := GVL_STATE.G_Flood_Warning[L_i];
    L_Runtime_State.Leak_Confirmed := GVL_STATE.G_Flood_Alarm[L_i];
    L_Runtime_State.Active_Safety_Leak_Latched := GVL_INTENT_SAFETY.I_Leak_Alarm_Active;
    L_Runtime_State.Active_Global_Close_Path := GVL_COMMAND_SHADOW.G_Close_Valve_35 OR GVL_COMMAND_SHADOW.G_Close_Valve_36;

    // Runtime topology is the authoritative mapping source here. It is updated
    // earlier in PRG_Water_Supervisory_Publication before leak projection runs.
    L_Group := UINT_TO_INT(GVL_Water_Topology_Config.G_Config_Record[L_i].Primary_Valve_Group_Id);
    L_Runtime_State.Mapping_Valid :=
        GVL_Water_Topology_Config.G_Config_Record[L_i].Config_Valid
        AND (L_Group >= 1)
        AND (L_Group <= GVL_CONSTANTS.C_MAX_FLOOD_VALVES);
    L_Runtime_State.Mapping_Missing := NOT L_Runtime_State.Mapping_Valid;

    IF L_Runtime_State.Mapping_Valid THEN
        L_Runtime_State.Valve_Group_Id := TO_UINT(L_Group);
        L_Runtime_State.Selective_Isolation_Possible := TRUE;
        L_Runtime_State.Fallback_Global_Isolation_Required := FALSE;
    ELSE
        L_Runtime_State.Valve_Group_Id := 0;
        L_Runtime_State.Selective_Isolation_Possible := FALSE;
        L_Runtime_State.Fallback_Global_Isolation_Required := TRUE;
    END_IF;

    L_Runtime_State.Logical_Sensor_Valid := TRUE;
    L_Runtime_State.Hydraulic_Zone_Id := TO_UINT(L_i);
    L_Runtime_State.Hydraulic_Segment_Id := GVL_Water_Topology_Config.G_Config_Record[L_i].Hydraulic_Segment_Id;
    L_Runtime_State.Isolation_Group_Id := L_Runtime_State.Valve_Group_Id;

    IF L_Runtime_State.Leak_Confirmed THEN
        L_Runtime_State.Leak_Confidence := 1.0;
    ELSIF L_Runtime_State.Leak_Warning_Active THEN
        L_Runtime_State.Leak_Confidence := 0.5;
    ELSE
        L_Runtime_State.Leak_Confidence := 0.0;
    END_IF;

    L_Runtime_State.Sensor_Quality_Valid := TRUE;

    IF L_Runtime_State.Leak_Confirmed THEN
        IF L_Runtime_State.Mapping_Valid THEN
            L_Runtime_State.Reason_Code := 1;
            L_Runtime_State.Reason_Text := 'Leak confirmed';
        ELSE
            L_Runtime_State.Reason_Code := 2;
            L_Runtime_State.Reason_Text := 'Leak confirmed fallback';
        END_IF;
    ELSIF L_Runtime_State.Leak_Warning_Active THEN
        L_Runtime_State.Reason_Code := 3;
        L_Runtime_State.Reason_Text := 'Leak warning active';
    ELSE
        L_Runtime_State.Reason_Code := 0;
        L_Runtime_State.Reason_Text := 'No leak activity';
    END_IF;

    L_Runtime_State.Warning_Started_Event := GVL_STATE.G_Flood_Warning_Rise[L_i];
    L_Runtime_State.Leak_Confirmed_Event := GVL_STATE.G_Flood_Alarm_Rise[L_i];
    L_Runtime_State.Leak_Cleared_Event := GVL_STATE.G_Flood_Alarm_Fall[L_i];
    L_Runtime_State.Isolation_Requested_Event := L_Runtime_State.Leak_Confirmed;
    L_Runtime_State.Mapping_Invalid_Event := L_Runtime_State.Mapping_Missing;
    L_Runtime_State.Supervisory_Observation_Only := TRUE;

    GVL_Water_Runtime_Projection.G_Leak_Runtime_State[L_i] := L_Runtime_State;

    L_Global_Leak := L_Global_Leak OR L_Runtime_State.Leak_Confirmed;
    L_Global_Warning := L_Global_Warning OR L_Runtime_State.Leak_Warning_Active;
END_FOR;

GVL_Water_Runtime_Projection.G_Global_Leak_Active := L_Global_Leak;
GVL_Water_Runtime_Projection.G_Global_Warning_Active := L_Global_Warning;
GVL_Water_Runtime_Projection.G_Projection_Valid := TRUE;
GVL_Water_Runtime_Projection.G_Last_Projection_MS := VI_System_Time_MS;
GVL_Water_Runtime_Projection.G_Runtime_Projection_Status_Code := 0;
GVL_Water_Runtime_Projection.G_Runtime_Projection_Status_Text := 'Water runtime semantic projection active';

END_FUNCTION_BLOCK

(* ---- FB_Water_Leakage_Manager.st ---- *)
FUNCTION_BLOCK FB_Water_Leakage_Manager
VAR_INPUT
    VI_System_Time_MS : UDINT;
    VI_IsActivePLC    : BOOL;
    VI_Config         : ST_Flood_Global_Config;
END_VAR

VAR_IN_OUT
    VI_Sensors : ARRAY[1..GVL_CONSTANTS.C_MAX_FLOOD_SENSORS] OF BOOL;
END_VAR

VAR_OUTPUT
    VO_Status_Msg     : STRING(200);

    // Health signals
    VO_Leak_Detected      : BOOL;
    VO_Leak_Warning_Level : BOOL;
END_VAR

VAR
    L_i             : INT;
    L_Sensor_Timers : ARRAY[1..GVL_CONSTANTS.C_MAX_FLOOD_SENSORS] OF FB_System_Timer;
    L_Any_Leak      : BOOL;
    L_Any_Warning   : BOOL;

    fbLeakLatch : RS;
END_VAR

IF NOT VI_IsActivePLC THEN RETURN; END_IF;

L_Any_Leak := FALSE;
L_Any_Warning := FALSE;

FOR L_i := 1 TO GVL_CONSTANTS.C_MAX_FLOOD_SENSORS DO
    L_Sensor_Timers[L_i](
        IN := VI_Sensors[L_i],
        PT := TO_TIME(VI_Config.min_duration_ms + VI_Config.warning_duration_ms),
        VI_System_Time_MS := VI_System_Time_MS
    );

    IF L_Sensor_Timers[L_i].ET >= TO_TIME(VI_Config.min_duration_ms) THEN
        L_Any_Warning := TRUE;

        IF L_Sensor_Timers[L_i].Q THEN
            L_Any_Leak := TRUE;
        END_IF;
    END_IF;
END_FOR;

// Latch аварии
fbLeakLatch(
    S := L_Any_Leak,
    R1 := GVL_INTENT_USER.I_Reset_Errors,
    Q => VO_Leak_Detected
);

VO_Leak_Warning_Level := L_Any_Warning;

// Status
IF VO_Leak_Detected THEN
    VO_Status_Msg := 'АВАРИЯ: ПРОТЕЧКА ВОДЫ.';
ELSIF L_Any_Warning THEN
    VO_Status_Msg := 'ПРЕДУПРЕЖДЕНИЕ: ОБНАРУЖЕНА ВОДА.';
ELSE
    VO_Status_Msg := 'Система контроля протечек в норме';
END_IF;
// >>> BULK_SYNC_ANCHOR: FB_Water_Leakage_Manager <<<

(* ---- FB_Water_Orchestration_Runtime.st ---- *)
FUNCTION_BLOCK FB_Water_Orchestration_Runtime
VAR_INPUT
    VI_Enable : BOOL;
    VI_System_Time_MS : UDINT;
END_VAR
VAR
    L_i : INT;

    L_Path : ST_Water_Isolation_Path_Runtime_State;
    L_Traversal : ST_Water_Graph_Traversal_State;
    L_Orchestration : ST_Water_Orchestration_Runtime_State;

    L_Any_Conflict : BOOL;
    L_Any_Escalation : BOOL;
END_VAR

IF NOT VI_Enable THEN
    GVL_Water_Orchestration.G_Runtime_Valid := FALSE;
    RETURN;
END_IF;

FOR L_i := 1 TO GVL_CONSTANTS.C_MAX_FLOOD_SENSORS DO

    L_Path :=
        GVL_Water_Hydraulic_Graph.G_Isolation_Path[L_i];

    // Traversal runtime.
    L_Traversal.Runtime_Valid := TRUE;

    L_Traversal.Runtime_System_Time_MS :=
        VI_System_Time_MS;

    L_Traversal.Sensor_Id := TO_UINT(L_i);

    L_Traversal.Start_Segment_Id :=
        L_Path.Active_Isolation_Group_Id;

    L_Traversal.Target_Valve_Group_Id :=
        L_Path.Active_Valve_Group_Id;

    L_Traversal.Shared_Trunk_Traversal :=
        L_Path.Shared_Trunk_Impact;

    L_Traversal.Upstream_Dependency_Detected :=
        L_Path.Shared_Trunk_Impact;

    L_Traversal.Downstream_Impact_Detected :=
        L_Path.Cross_Zone_Impact;

    L_Traversal.Traversal_Valid :=
        L_Path.Isolation_Path_Valid;

    L_Traversal.Traversal_Conflict :=
        L_Path.Conflict_Detected;

    L_Traversal.Traversal_Ambiguous :=
        L_Path.Isolation_Path_Ambiguous;

    IF L_Path.Multi_Valve_Path THEN
        L_Traversal.Dependency_Depth := 2;
    ELSE
        L_Traversal.Dependency_Depth := 1;
    END_IF;

    L_Traversal.Selective_Path_Allowed :=
        L_Path.Selective_Isolation_Allowed;

    L_Traversal.Global_Fallback_Required :=
        L_Path.Global_Fallback_Required;

    // Orchestration runtime.
    L_Orchestration.Runtime_Valid := TRUE;

    L_Orchestration.Runtime_System_Time_MS :=
        VI_System_Time_MS;

    L_Orchestration.Isolation_Sequence_Active :=
        L_Traversal.Traversal_Valid;

    L_Orchestration.Shared_Trunk_Sequencing :=
        L_Traversal.Shared_Trunk_Traversal;

    L_Orchestration.Staged_Close_Required :=
        L_Path.Multi_Valve_Path;

    L_Orchestration.Recovery_Sequence_Active :=
        GVL_INTENT_SAFETY.I_Water_Selective_Recovery_Allowed;

    L_Orchestration.Staged_Open_Required :=
        L_Orchestration.Recovery_Sequence_Active
        AND L_Path.Multi_Valve_Path;

    L_Orchestration.Observation_Window_Active :=
        L_Orchestration.Recovery_Sequence_Active;

    // Conservative sequencing governance.
    IF L_Traversal.Traversal_Conflict
       OR L_Traversal.Traversal_Ambiguous THEN

        L_Orchestration.Rollback_Required := TRUE;
        L_Orchestration.Escalation_Required := TRUE;
        L_Orchestration.Sequencing_Valid := FALSE;

        L_Orchestration.Status_Code := 2;
        L_Orchestration.Status_Text :=
            'Orchestration conflict escalation active';

    ELSE

        L_Orchestration.Sequencing_Valid := TRUE;

        IF L_Orchestration.Shared_Trunk_Sequencing THEN
            L_Orchestration.Status_Code := 1;
            L_Orchestration.Status_Text :=
                'Shared trunk orchestration active';
        ELSE
            L_Orchestration.Status_Code := 0;
            L_Orchestration.Status_Text :=
                'Deterministic orchestration active';
        END_IF;

    END_IF;

    GVL_Water_Orchestration.G_Traversal_State[L_i] :=
        L_Traversal;

    GVL_Water_Orchestration.G_Orchestration_State[L_i] :=
        L_Orchestration;

    L_Any_Conflict :=
        L_Any_Conflict
        OR L_Traversal.Traversal_Conflict;

    L_Any_Escalation :=
        L_Any_Escalation
        OR L_Orchestration.Escalation_Required;

END_FOR;

GVL_Water_Orchestration.G_Topology_Version := 1;
GVL_Water_Orchestration.G_Config_Runtime_Ready := TRUE;

GVL_Water_Orchestration.G_Any_Traversal_Conflict :=
    L_Any_Conflict;

GVL_Water_Orchestration.G_Any_Escalation_Required :=
    L_Any_Escalation;

GVL_Water_Orchestration.G_Runtime_Valid := TRUE;
GVL_Water_Orchestration.G_Last_Update_MS := VI_System_Time_MS;

IF L_Any_Escalation THEN
    GVL_Water_Orchestration.G_Status_Code := 2;
    GVL_Water_Orchestration.G_Status_Text :=
        'Water orchestration escalation active';
ELSIF L_Any_Conflict THEN
    GVL_Water_Orchestration.G_Status_Code := 1;
    GVL_Water_Orchestration.G_Status_Text :=
        'Water orchestration conflict detected';
ELSE
    GVL_Water_Orchestration.G_Status_Code := 0;
    GVL_Water_Orchestration.G_Status_Text :=
        'Water orchestration runtime healthy';
END_IF;

END_FUNCTION_BLOCK

(* ---- FB_Water_Output_Projection.st ---- *)
FUNCTION_BLOCK FB_Water_Output_Projection
VAR_INPUT
    VI_Zone_Enable : ARRAY[1..GVL_CONSTANTS.C_MAX_WATER_ZONES] OF BOOL;
    VI_Valve_35_Close : BOOL;
    VI_Valve_36_Close : BOOL;
END_VAR
VAR
    L_i : INT;
END_VAR

FOR L_i := 1 TO GVL_CONSTANTS.C_MAX_WATER_ZONES DO
    GVL_WATER_OUTPUT.DO_Water_Zone_Enable[L_i] := VI_Zone_Enable[L_i];
END_FOR;

GVL_WATER_OUTPUT.DO_Water_Valve_35_Close := VI_Valve_35_Close;
GVL_WATER_OUTPUT.DO_Water_Valve_36_Close := VI_Valve_36_Close;

END_FUNCTION_BLOCK
// >>> BULK_SYNC_ANCHOR: FB_Water_Output_Projection <<<

(* ---- FB_Water_Output_Projector.st ---- *)
FUNCTION_BLOCK FB_Water_Output_Projector
VAR_INPUT
    VI_Enable : BOOL;
    VI_System_Time_MS : UDINT;
END_VAR
VAR
    L_i : INT;
    L_Authority : ST_Water_Isolation_Authority_State;
    L_Valve : ST_Water_Valve_Runtime_State;
    L_Output : ST_Water_Output_Projection_State;
    L_Any_Projected : BOOL;
    L_Any_Denied : BOOL;
    L_Global_Fallback : BOOL;
END_VAR

IF NOT VI_Enable THEN
    GVL_Water_Output_Projection.G_Runtime_Valid := FALSE;
    RETURN;
END_IF;

L_Any_Projected := FALSE;
L_Any_Denied := FALSE;
L_Global_Fallback := FALSE;

FOR L_i := 1 TO GVL_CONSTANTS.C_MAX_FLOOD_SENSORS DO

    L_Authority := GVL_Water_Isolation_Authority.G_Authority_State[L_i];
    L_Valve := GVL_Water_Valve_Runtime.G_Valve_Runtime_State[L_i];

    L_Output.Projection_Valid := FALSE;
    L_Output.Projection_Valid := TRUE;
    L_Output.Projection_System_Time_MS := VI_System_Time_MS;
    L_Output.Output_Owner_Valid := TRUE;
    L_Output.Output_Owner_Id := TO_UINT(L_i);
    L_Output.Valve_Id := L_Valve.Valve_Id;
    L_Output.Valve_Group_Id := L_Valve.Valve_Group_Id;
    L_Output.Selective_Authority_Allowed := L_Authority.Selective_Authority_Allowed;
    L_Output.Global_Fallback_Required := L_Authority.Global_Fallback_Required;
    L_Output.Authority_Valid := L_Authority.Decision_Valid;

    IF L_Output.Global_Fallback_Required THEN
        L_Output.Projection_Allowed := TRUE;
        L_Output.Physical_Close_Project := TRUE;
        L_Output.Expected_Closed := TRUE;
        L_Output.Projection_Code := 1;
        L_Output.Projection_Text := 'Global fallback output projection active';
        L_Global_Fallback := TRUE;
    ELSIF L_Output.Selective_Authority_Allowed AND L_Output.Authority_Valid THEN
        L_Output.Projection_Allowed := TRUE;
        L_Output.Physical_Close_Project := TRUE;
        L_Output.Expected_Closed := TRUE;
        L_Output.Projection_Code := 10;
        L_Output.Projection_Text := 'Selective authority output projection active';
    ELSE
        L_Output.Projection_Denied := TRUE;
        L_Output.Projection_Code := 100;
        L_Output.Projection_Text := 'Projection denied';
        L_Any_Denied := TRUE;
    END_IF;

    L_Output.Confirmed_Closed := L_Valve.Confirmed_Closed;
    L_Output.Confirmed_Open := L_Valve.Confirmed_Open;
    L_Output.Confirmation_Unknown := L_Valve.Confirmation_Unknown;
    L_Output.Projection_Activated_Event := L_Output.Projection_Allowed;
    L_Output.Projection_Denied_Event := L_Output.Projection_Denied;

    GVL_Water_Output_Projection.G_Output_Projection_State[L_i] := L_Output;
    L_Any_Projected := L_Any_Projected OR L_Output.Projection_Allowed;
END_FOR;

GVL_Water_Output_Projection.G_Any_Output_Projected := L_Any_Projected;
GVL_Water_Output_Projection.G_Any_Projection_Denied := L_Any_Denied;
GVL_Water_Output_Projection.G_Global_Fallback_Projecting := L_Global_Fallback;
GVL_Water_Output_Projection.G_Runtime_Valid := TRUE;
GVL_Water_Output_Projection.G_Last_Update_MS := VI_System_Time_MS;

IF L_Global_Fallback THEN
    GVL_Water_Output_Projection.G_Status_Code := 2;
    GVL_Water_Output_Projection.G_Status_Text := 'Global fallback output projection active';
ELSIF L_Any_Projected THEN
    GVL_Water_Output_Projection.G_Status_Code := 1;
    GVL_Water_Output_Projection.G_Status_Text := 'Selective output projection active';
ELSE
    GVL_Water_Output_Projection.G_Status_Code := 0;
    GVL_Water_Output_Projection.G_Status_Text := 'No output projections active';
END_IF;

END_FUNCTION_BLOCK

(* ---- FB_Water_Output_Reconciliation.st ---- *)
FUNCTION_BLOCK FB_Water_Output_Reconciliation
VAR_INPUT
    VI_Enable : BOOL;
    VI_System_Time_MS : UDINT;
END_VAR
VAR
    L_i : INT;
    L_Output : ST_Water_Output_Projection_State;
    L_Valve : ST_Water_Valve_Runtime_State;
    L_State : ST_Water_Output_Reconciliation_State;
    L_Any_Runtime_Mismatch : BOOL;
    L_Any_Confirmation_Mismatch : BOOL;
    L_Any_Conflict : BOOL;
END_VAR

IF NOT VI_Enable THEN
    GVL_Water_Output_Reconciliation.G_Runtime_Valid := FALSE;
    RETURN;
END_IF;

FOR L_i := 1 TO GVL_CONSTANTS.C_MAX_FLOOD_SENSORS DO

    L_Output := GVL_Water_Output_Projection.G_Output_Projection_State[L_i];
    L_Valve := GVL_Water_Valve_Runtime.G_Valve_Runtime_State[L_i];

    L_State.Runtime_Valid := TRUE;
    L_State.Runtime_System_Time_MS := VI_System_Time_MS;

    L_State.Valve_Group_Id := L_Output.Valve_Group_Id;
    L_State.Projection_Active := L_Output.Physical_Close_Project;
    L_State.Runtime_Output_Active := L_Valve.Physical_Output_Active;
    L_State.Expected_Closed := L_Output.Expected_Closed;
    L_State.Confirmed_Closed := L_Valve.Confirmed_Closed;
    L_State.Feedback_Invalid := L_Valve.Feedback_Invalid;

    IF L_Valve.Confirmation_Available THEN

        IF L_State.Projection_Active <> L_State.Runtime_Output_Active THEN
            L_State.Projection_Runtime_Mismatch := TRUE;
        END_IF;

        IF L_State.Expected_Closed
           AND NOT L_State.Confirmed_Closed THEN
            L_State.Projection_Confirmation_Mismatch := TRUE;
        END_IF;

    END_IF;

    IF L_Output.Projection_Allowed
       AND L_Output.Projection_Denied THEN
        L_State.Conflict_Detected := TRUE;
    END_IF;

    IF L_Output.Valve_Group_Id = 0 THEN
        L_State.Topology_Invalid := TRUE;
    END_IF;

    L_State.Reconciliation_Healthy :=
        NOT L_State.Projection_Runtime_Mismatch
        AND NOT L_State.Projection_Confirmation_Mismatch
        AND NOT L_State.Conflict_Detected
        AND NOT L_State.Topology_Invalid;

    IF L_State.Conflict_Detected THEN
        L_State.Status_Code := 3;
        L_State.Status_Text := 'Projection conflict detected';
    ELSIF L_State.Projection_Runtime_Mismatch THEN
        L_State.Status_Code := 2;
        L_State.Status_Text := 'Projection runtime mismatch';
    ELSIF L_State.Projection_Confirmation_Mismatch THEN
        L_State.Status_Code := 1;
        L_State.Status_Text := 'Projection confirmation mismatch';
    ELSE
        L_State.Status_Code := 0;
        L_State.Status_Text := 'Reconciliation healthy';
    END_IF;

    GVL_Water_Output_Reconciliation.G_Reconciliation_State[L_i] := L_State;
END_FOR;

END_FUNCTION_BLOCK

(* ---- FB_Water_Physical_Runtime.st ---- *)
FUNCTION_BLOCK FB_Water_Physical_Runtime
VAR_INPUT
    VI_Enable : BOOL;
    VI_System_Time_MS : UDINT;
END_VAR
VAR
    L_i : INT;
    L_Output : ST_Water_Output_Projection_State;
    L_Feedback : ST_Water_Valve_Feedback_State;
    L_Convergence : ST_Water_Physical_Convergence_State;
    L_Diagnostics : ST_Water_Actuator_Diagnostics_State;
    L_Any_Convergence_Degraded : BOOL;
    L_Any_Diagnostics_Degraded : BOOL;
    L_Any_Escalation : BOOL;
END_VAR

IF NOT VI_Enable THEN
    GVL_Water_Physical_Runtime.G_Runtime_Valid := FALSE;
    RETURN;
END_IF;

FOR L_i := 1 TO GVL_CONSTANTS.C_MAX_FLOOD_SENSORS DO
    L_Output := GVL_Water_Output_Projection.G_Output_Projection_State[L_i];
    L_Feedback := GVL_Water_Valve_Feedback.G_Valve_Feedback_State[L_i];

    L_Convergence.Runtime_Valid := TRUE;
    L_Convergence.Runtime_System_Time_MS := VI_System_Time_MS;
    L_Convergence.Sensor_Id := TO_UINT(L_i);
    L_Convergence.Projection_Active := L_Output.Projection_Allowed;
    L_Convergence.Physical_Open_Confirmed := L_Feedback.Confirmed_Open;
    L_Convergence.Physical_Closed_Confirmed := L_Feedback.Confirmed_Closed;
    L_Convergence.Physical_State_Confirmed := L_Feedback.Confirmed_Open OR L_Feedback.Confirmed_Closed;

    IF L_Feedback.Feedback_Available THEN
        IF L_Output.Expected_Closed AND NOT L_Feedback.Confirmed_Closed THEN
            L_Convergence.Projection_Mismatch := TRUE;
            L_Convergence.Physical_Mismatch := TRUE;
        END_IF;

        IF NOT L_Convergence.Projection_Mismatch AND NOT L_Feedback.Feedback_Timeout THEN
            L_Convergence.Runtime_Converged := TRUE;
        END_IF;
    ELSE
        L_Convergence.Runtime_Mismatch := FALSE;
    END_IF;

    IF L_Convergence.Projection_Mismatch OR L_Feedback.Feedback_Conflict THEN
        L_Convergence.Convergence_Degraded := TRUE;
        L_Convergence.Escalation_Required := TRUE;
        L_Convergence.Status_Code := 2;
        L_Convergence.Status_Text := 'Physical convergence mismatch detected';
    ELSIF L_Convergence.Runtime_Converged THEN
        L_Convergence.Status_Code := 1;
        L_Convergence.Status_Text := 'Physical runtime converged';
    ELSE
        L_Convergence.Status_Code := 0;
        L_Convergence.Status_Text := 'Physical convergence observe-only';
    END_IF;

    L_Diagnostics.Runtime_Valid := TRUE;
    L_Diagnostics.Runtime_System_Time_MS := VI_System_Time_MS;
    L_Diagnostics.Valve_Group_Id := L_Output.Valve_Group_Id;
    L_Diagnostics.Travel_Active := L_Output.Projection_Allowed AND L_Feedback.Feedback_Available AND NOT L_Convergence.Runtime_Converged;

    IF L_Diagnostics.Travel_Active THEN
        L_Diagnostics.Travel_Time_MS := 100;
    ELSE
        L_Diagnostics.Travel_Time_MS := 0;
    END_IF;

    IF L_Diagnostics.Travel_Time_MS > 4000 THEN
        L_Diagnostics.Travel_Timeout := TRUE;
        L_Diagnostics.Stuck_Suspected := TRUE;
    END_IF;

    IF L_Diagnostics.Travel_Timeout THEN
        L_Diagnostics.Diagnostics_Degraded := TRUE;
        L_Diagnostics.Escalation_Required := TRUE;
        L_Diagnostics.Failure_Count := 1;
        L_Diagnostics.Status_Code := 2;
        L_Diagnostics.Status_Text := 'Actuator travel timeout detected';
    ELSE
        L_Diagnostics.Status_Code := 0;
        L_Diagnostics.Status_Text := 'Actuator diagnostics healthy';
    END_IF;

    GVL_Water_Physical_Runtime.G_Convergence_State[L_i] := L_Convergence;
    GVL_Water_Physical_Runtime.G_Actuator_Diagnostics[L_i] := L_Diagnostics;

    L_Any_Convergence_Degraded := L_Any_Convergence_Degraded OR L_Convergence.Convergence_Degraded;
    L_Any_Diagnostics_Degraded := L_Any_Diagnostics_Degraded OR L_Diagnostics.Diagnostics_Degraded;
    L_Any_Escalation := L_Any_Escalation OR L_Convergence.Escalation_Required OR L_Diagnostics.Escalation_Required;
END_FOR;

GVL_Water_Physical_Runtime.G_Any_Convergence_Degraded := L_Any_Convergence_Degraded;
GVL_Water_Physical_Runtime.G_Any_Diagnostics_Degraded := L_Any_Diagnostics_Degraded;
GVL_Water_Physical_Runtime.G_Any_Escalation_Required := L_Any_Escalation;
GVL_Water_Physical_Runtime.G_Runtime_Valid := TRUE;
GVL_Water_Physical_Runtime.G_Last_Update_MS := VI_System_Time_MS;

IF L_Any_Escalation THEN
    GVL_Water_Physical_Runtime.G_Status_Code := 2;
    GVL_Water_Physical_Runtime.G_Status_Text := 'Physical runtime escalation active';
ELSIF L_Any_Convergence_Degraded THEN
    GVL_Water_Physical_Runtime.G_Status_Code := 1;
    GVL_Water_Physical_Runtime.G_Status_Text := 'Physical convergence degraded';
ELSE
    GVL_Water_Physical_Runtime.G_Status_Code := 0;
    GVL_Water_Physical_Runtime.G_Status_Text := 'Physical runtime healthy';
END_IF;

END_FUNCTION_BLOCK

(* ---- FB_Water_Recovery_Runtime.st ---- *)
FUNCTION_BLOCK FB_Water_Recovery_Runtime
VAR_INPUT
    VI_Enable : BOOL;
    VI_System_Time_MS : UDINT;
END_VAR
VAR
    L_i : INT;
    L_Feedback : ST_Water_Valve_Feedback_State;
    L_State : ST_Water_Recovery_Runtime_State;
    L_Any_Denied : BOOL;
    L_Any_Unsafe : BOOL;
END_VAR

IF NOT VI_Enable THEN
    GVL_Water_Recovery_Runtime.G_Runtime_Valid := FALSE;
    RETURN;
END_IF;

L_Any_Denied := FALSE;
L_Any_Unsafe := FALSE;

FOR L_i := 1 TO GVL_CONSTANTS.C_MAX_FLOOD_SENSORS DO
    L_Feedback := GVL_Water_Valve_Feedback.G_Valve_Feedback_State[L_i];

    L_State.Runtime_Valid := FALSE;
    L_State.Runtime_System_Time_MS := 0;
    L_State.Recovery_Requested := FALSE;
    L_State.Recovery_Allowed := FALSE;
    L_State.Recovery_Denied := FALSE;
    L_State.Observation_Window_Active := FALSE;
    L_State.Unsafe_Recovery_Detected := FALSE;
    L_State.Valve_Degraded := FALSE;
    L_State.Confirmation_Healthy := FALSE;
    L_State.Recovery_Target_Valid := FALSE;
    L_State.Status_Code := 0;
    L_State.Status_Text := '';

    L_State.Runtime_Valid := TRUE;
    L_State.Runtime_System_Time_MS := VI_System_Time_MS;
    L_State.Recovery_Requested := GVL_INTENT_SAFETY.I_Water_Selective_Recovery_Allowed;
    L_State.Valve_Degraded := L_Feedback.Valve_Degraded;
    L_State.Confirmation_Healthy := NOT L_Feedback.Feedback_Conflict;
    L_State.Recovery_Target_Valid := L_Feedback.Valve_Group_Id <> 0;

    IF NOT L_State.Recovery_Requested THEN
        L_State.Status_Code := 0;
        L_State.Status_Text := 'Recovery observe only';
    ELSIF NOT L_State.Recovery_Target_Valid THEN
        L_State.Recovery_Denied := TRUE;
        L_State.Status_Code := 1;
        L_State.Status_Text := 'Recovery target invalid';
    ELSIF L_State.Valve_Degraded THEN
        L_State.Recovery_Denied := TRUE;
        L_State.Unsafe_Recovery_Detected := TRUE;
        L_State.Status_Code := 2;
        L_State.Status_Text := 'Recovery blocked by valve state';
    ELSIF NOT L_State.Confirmation_Healthy THEN
        L_State.Recovery_Denied := TRUE;
        L_State.Status_Code := 3;
        L_State.Status_Text := 'Recovery blocked by confirmation state';
    ELSE
        L_State.Recovery_Allowed := TRUE;
        L_State.Observation_Window_Active := TRUE;
        L_State.Status_Code := 0;
        L_State.Status_Text := 'Recovery governance healthy';
    END_IF;

    GVL_Water_Recovery_Runtime.G_Recovery_State[L_i] := L_State;
    L_Any_Denied := L_Any_Denied OR L_State.Recovery_Denied;
    L_Any_Unsafe := L_Any_Unsafe OR L_State.Unsafe_Recovery_Detected;
END_FOR;

GVL_Water_Recovery_Runtime.G_Any_Recovery_Denied := L_Any_Denied;
GVL_Water_Recovery_Runtime.G_Any_Unsafe_Recovery := L_Any_Unsafe;
GVL_Water_Recovery_Runtime.G_Runtime_Valid := TRUE;
GVL_Water_Recovery_Runtime.G_Last_Update_MS := VI_System_Time_MS;

IF L_Any_Unsafe THEN
    GVL_Water_Recovery_Runtime.G_Status_Code := 2;
    GVL_Water_Recovery_Runtime.G_Status_Text := 'Recovery risk detected';
ELSIF L_Any_Denied THEN
    GVL_Water_Recovery_Runtime.G_Status_Code := 1;
    GVL_Water_Recovery_Runtime.G_Status_Text := 'Recovery governance denied';
ELSIF GVL_INTENT_SAFETY.I_Water_Selective_Recovery_Allowed THEN
    GVL_Water_Recovery_Runtime.G_Status_Code := 0;
    GVL_Water_Recovery_Runtime.G_Status_Text := 'Recovery governance healthy';
ELSE
    GVL_Water_Recovery_Runtime.G_Status_Code := 0;
    GVL_Water_Recovery_Runtime.G_Status_Text := 'Recovery observe only';
END_IF;

END_FUNCTION_BLOCK

(* ---- FB_Water_Runtime_Hardening.st ---- *)
FUNCTION_BLOCK FB_Water_Runtime_Hardening
VAR_INPUT
    VI_Enable : BOOL;
    VI_System_Time_MS : UDINT;
END_VAR
VAR
    L_i : INT;

    L_FSM : ST_Water_Recovery_FSM_State;
    L_Event : ST_Water_Event_Log_Record;

    L_Any_Rollback : BOOL;
    L_Any_Escalation : BOOL;
END_VAR

IF NOT VI_Enable THEN
    GVL_Water_Runtime_Hardening.G_Runtime_Valid := FALSE;
    RETURN;
END_IF;

FOR L_i := 1 TO GVL_CONSTANTS.C_MAX_FLOOD_SENSORS DO

    // Recovery FSM.
    L_FSM.Runtime_Valid := TRUE;

    L_FSM.Runtime_System_Time_MS :=
        VI_System_Time_MS;

    L_FSM.Recovery_Domain_Id :=
        GVL_Water_Topology_Config.G_Config_Record[L_i].Recovery_Domain_Id;

    L_FSM.Recovery_Requested :=
        GVL_INTENT_SAFETY.I_Water_Selective_Recovery_Allowed;

    L_FSM.Recovery_Sequencing_Active :=
        GVL_Water_Orchestration.G_Orchestration_State[L_i].Recovery_Sequence_Active;

    L_FSM.Recovery_Verification_Window_Active :=
        GVL_Water_Orchestration.G_Orchestration_State[L_i].Observation_Window_Active;

    // Conservative runtime hardening.
    IF GVL_Water_Physical_Runtime.G_Convergence_State[L_i].Escalation_Required THEN

        L_FSM.Rollback_Required := TRUE;
        L_FSM.Escalation_Required := TRUE;
        L_FSM.Operator_Ack_Required := TRUE;
        L_FSM.Recovery_Denied := TRUE;
        L_FSM.FSM_State := 100;

        L_FSM.Status_Code := 2;
        L_FSM.Status_Text :=
            'Recovery rollback escalation active';

    ELSIF L_FSM.Recovery_Requested THEN

        L_FSM.Recovery_Completed := TRUE;
        L_FSM.FSM_State := 10;

        L_FSM.Status_Code := 1;
        L_FSM.Status_Text :=
            'Recovery sequencing active';

    ELSE

        L_FSM.FSM_State := 0;

        L_FSM.Status_Code := 0;
        L_FSM.Status_Text :=
            'Recovery FSM idle';

    END_IF;

    GVL_Water_Runtime_Hardening.G_Recovery_FSM[L_i] :=
        L_FSM;

    // Runtime event publication.
    IF L_i <= 128 THEN

        L_Event.Runtime_Valid := TRUE;

        L_Event.Event_Time_MS := VI_System_Time_MS;
        L_Event.Event_Id := TO_UINT(L_i);

        IF L_FSM.Escalation_Required THEN
            L_Event.Event_Text :=
                'Water runtime escalation active';
        ELSE
            L_Event.Event_Text :=
                'Water runtime healthy';
        END_IF;

        GVL_Water_Runtime_Hardening.G_Event_Log[L_i] :=
            L_Event;

    END_IF;

    L_Any_Rollback :=
        L_Any_Rollback
        OR L_FSM.Rollback_Required;

    L_Any_Escalation :=
        L_Any_Escalation
        OR L_FSM.Escalation_Required;

END_FOR;

GVL_Water_Runtime_Hardening.G_Runtime_Quarantine_Active :=
    L_Any_Escalation;

GVL_Water_Runtime_Hardening.G_Service_Mode_Active := FALSE;
GVL_Water_Runtime_Hardening.G_Maintenance_Mode_Active := FALSE;

GVL_Water_Runtime_Hardening.G_Any_Rollback_Required :=
    L_Any_Rollback;

GVL_Water_Runtime_Hardening.G_Any_Escalation_Required :=
    L_Any_Escalation;

GVL_Water_Runtime_Hardening.G_Runtime_Valid := TRUE;
GVL_Water_Runtime_Hardening.G_Last_Update_MS := VI_System_Time_MS;

IF L_Any_Escalation THEN
    GVL_Water_Runtime_Hardening.G_Status_Code := 2;
    GVL_Water_Runtime_Hardening.G_Status_Text :=
        'Runtime quarantine escalation active';
ELSIF L_Any_Rollback THEN
    GVL_Water_Runtime_Hardening.G_Status_Code := 1;
    GVL_Water_Runtime_Hardening.G_Status_Text :=
        'Recovery rollback active';
ELSE
    GVL_Water_Runtime_Hardening.G_Status_Code := 0;
    GVL_Water_Runtime_Hardening.G_Status_Text :=
        'Production runtime hardening active';
END_IF;

END_FUNCTION_BLOCK

(* ---- FB_Water_Topology_Config_Runtime.st ---- *)
FUNCTION_BLOCK FB_Water_Topology_Config_Runtime
VAR_INPUT
    VI_Enable : BOOL;
    VI_System_Time_MS : UDINT;
END_VAR
VAR
    L_i : INT;
    L_Config : ST_Water_Topology_Config_Record;
    L_Any_Invalid : BOOL;
    L_Any_Multi_Valve : BOOL;
    L_Default_Group : UINT;
END_VAR

IF NOT VI_Enable THEN
    GVL_Water_Topology_Config.G_Runtime_Valid := FALSE;
    RETURN;
END_IF;

L_Any_Invalid := FALSE;
L_Any_Multi_Valve := FALSE;

FOR L_i := 1 TO GVL_CONSTANTS.C_MAX_FLOOD_SENSORS DO

    L_Config := GVL_Water_Topology_Config_Source.G_Source_Record[L_i];
    L_Default_Group := 0;

    // Default topology from current TZ:
    // sensors 1..2   -> zone 1 kitchen, valves 1/2;
    // sensors 3..4   -> zone 2 master bathroom, valves 3/4;
    // sensors 5..9   -> zone 3 guest bathrooms + laundry, valves 5/6;
    // sensors 10..12 -> zone 4 boiler/common inlet, valves 35/36.
    IF (L_i >= 1) AND (L_i <= 2) THEN
        L_Default_Group := 1;
    ELSIF (L_i >= 3) AND (L_i <= 4) THEN
        L_Default_Group := 2;
    ELSIF (L_i >= 5) AND (L_i <= 9) THEN
        L_Default_Group := 3;
    ELSIF (L_i >= 10) AND (L_i <= 12) THEN
        L_Default_Group := 4;
    END_IF;

    IF NOT L_Config.Config_Valid THEN
        L_Config.Config_Valid := L_Default_Group <> 0;
        L_Config.Config_Version := 1;
        L_Config.Sensor_Id := TO_UINT(L_i);
        L_Config.Logical_Zone_Id := TO_UINT(L_i);
        L_Config.Hydraulic_Segment_Id := L_Default_Group;
        L_Config.Isolation_Group_Id := L_Default_Group;
        L_Config.Primary_Valve_Group_Id := L_Default_Group;
        L_Config.Secondary_Valve_Group_Id := 0;
        L_Config.Fallback_Domain_Id := 4;
        L_Config.Recovery_Domain_Id := L_Default_Group;
        L_Config.Shared_Trunk := L_Default_Group = 4;
        L_Config.Cross_Zone_Dependency := L_Default_Group = 4;
        L_Config.Multi_Valve_Required := L_Default_Group <> 0;
        L_Config.Recovery_Requires_Manual_Ack := TRUE;
    END_IF;

    IF (NOT L_Config.Config_Valid)
       OR (L_Config.Primary_Valve_Group_Id < 1)
       OR (L_Config.Primary_Valve_Group_Id > 4) THEN
        L_Config.Config_Valid := FALSE;
        L_Config.Status_Code := 1;
        L_Config.Status_Text := 'Invalid water topology config';
    ELSE
        L_Config.Status_Code := 0;
        CASE L_Config.Primary_Valve_Group_Id OF
            1:
                L_Config.Status_Text := 'Topology loaded: zone 1 kitchen valves 1/2';
            2:
                L_Config.Status_Text := 'Topology loaded: zone 2 master bathroom valves 3/4';
            3:
                L_Config.Status_Text := 'Topology loaded: zone 3 guest bathrooms + laundry valves 5/6';
            4:
                L_Config.Status_Text := 'Topology loaded: zone 4 boiler/common inlet 35/36';
        ELSE
                L_Config.Status_Text := 'Topology loaded';
        END_CASE;
    END_IF;

    GVL_Water_Topology_Config.G_Config_Record[L_i] := L_Config;

    L_Any_Invalid := L_Any_Invalid OR NOT L_Config.Config_Valid;
    L_Any_Multi_Valve := L_Any_Multi_Valve OR L_Config.Multi_Valve_Required;

END_FOR;

GVL_Water_Topology_Config.G_Active_Config_Version := GVL_Water_Topology_Config_Source.G_Source_Version;
GVL_Water_Topology_Config.G_Config_Loaded := TRUE;
GVL_Water_Topology_Config.G_Runtime_Remap_Ready := TRUE;
GVL_Water_Topology_Config.G_Any_Invalid_Config := L_Any_Invalid;
GVL_Water_Topology_Config.G_Any_Multi_Valve_Required := L_Any_Multi_Valve;
GVL_Water_Topology_Config.G_Runtime_Valid := NOT L_Any_Invalid;
GVL_Water_Topology_Config.G_Last_Update_MS := VI_System_Time_MS;

IF L_Any_Invalid THEN
    GVL_Water_Topology_Config.G_Status_Code := 2;
    GVL_Water_Topology_Config.G_Status_Text := 'Topology config invalid';
ELSIF L_Any_Multi_Valve THEN
    GVL_Water_Topology_Config.G_Status_Code := 1;
    GVL_Water_Topology_Config.G_Status_Text := 'Multi-valve topology active';
ELSE
    GVL_Water_Topology_Config.G_Status_Code := 0;
    GVL_Water_Topology_Config.G_Status_Text := 'Topology config runtime healthy';
END_IF;

END_FUNCTION_BLOCK

(* ---- FB_Water_Valve_Feedback_Runtime.st ---- *)
FUNCTION_BLOCK FB_Water_Valve_Feedback_Runtime
VAR_INPUT
    VI_Enable : BOOL;
    VI_System_Time_MS : UDINT;
END_VAR
VAR
    L_i : INT;
    L_State : ST_Water_Valve_Feedback_State;
    L_Empty_State : ST_Water_Valve_Feedback_State;
    L_Any_Degraded : BOOL;
    L_Any_Timeout : BOOL;
    L_Any_Conflict : BOOL;
    L_Command_Open : BOOL;
    L_Command_Close : BOOL;
    L_Command_Active : BOOL;
    L_Desired_Code : USINT;
    L_Elapsed_MS : UDINT;
    L_Command_Start_MS : ARRAY[1..8] OF UDINT;
    L_Prev_Desired_Code : ARRAY[1..8] OF USINT;
END_VAR

IF NOT VI_Enable THEN
    GVL_Water_Valve_Feedback.G_Runtime_Valid := FALSE;
    RETURN;
END_IF;

L_Any_Degraded := FALSE;
L_Any_Timeout := FALSE;
L_Any_Conflict := FALSE;

FOR L_i := 1 TO 8 DO
    L_State := L_Empty_State;
    L_State.Runtime_Valid := TRUE;
    L_State.Runtime_System_Time_MS := VI_System_Time_MS;

    // Valve identity used by HMI/diagnostics:
    // 1..6 = local riser valves, 7 = common inlet 35, 8 = common inlet 36.
    L_State.Valve_Group_Id := TO_UINT(L_i);
    L_State.Feedback_Available := TRUE;

    CASE L_i OF
        1..6:
            L_Command_Open := GVL_WATER_OUTPUT.DO_Water_Local_Valve_Open[L_i];
            L_Command_Close := GVL_WATER_OUTPUT.DO_Water_Local_Valve_Close[L_i];
        7:
            L_Command_Open := GVL_WATER_OUTPUT.DO_Water_Valve_35_Open;
            L_Command_Close := GVL_WATER_OUTPUT.DO_Water_Valve_35_Close;
        8:
            L_Command_Open := GVL_WATER_OUTPUT.DO_Water_Valve_36_Open;
            L_Command_Close := GVL_WATER_OUTPUT.DO_Water_Valve_36_Close;
    ELSE
            L_Command_Open := FALSE;
            L_Command_Close := FALSE;
    END_CASE;

    L_State.Physical_Open_Feedback := GVL_STATE.G_Water_Zone_Open_FB[L_i];
    L_State.Physical_Closed_Feedback := GVL_STATE.G_Water_Zone_Close_FB[L_i];

    IF L_State.Physical_Open_Feedback AND L_State.Physical_Closed_Feedback THEN
        L_State.Feedback_Conflict := TRUE;
        L_State.Feedback_Invalid := TRUE;
        L_State.Valve_Degraded := TRUE;
    END_IF;

    L_State.Confirmed_Open := L_State.Physical_Open_Feedback AND NOT L_State.Physical_Closed_Feedback;
    L_State.Confirmed_Closed := L_State.Physical_Closed_Feedback AND NOT L_State.Physical_Open_Feedback;
    L_State.Confirmation_Unknown := NOT L_State.Confirmed_Open AND NOT L_State.Confirmed_Closed AND NOT L_State.Feedback_Conflict;

    IF L_Command_Close AND NOT L_Command_Open THEN
        L_Desired_Code := 2;
    ELSIF L_Command_Open AND NOT L_Command_Close THEN
        L_Desired_Code := 1;
    ELSE
        L_Desired_Code := 0;
    END_IF;

    IF L_Desired_Code <> L_Prev_Desired_Code[L_i] THEN
        L_Command_Start_MS[L_i] := VI_System_Time_MS;
        L_Prev_Desired_Code[L_i] := L_Desired_Code;
    END_IF;

    L_Command_Active := (L_Desired_Code <> 0);

    IF L_Command_Active THEN
        IF VI_System_Time_MS >= L_Command_Start_MS[L_i] THEN
            L_Elapsed_MS := VI_System_Time_MS - L_Command_Start_MS[L_i];
        ELSE
            L_Elapsed_MS := (4294967295 - L_Command_Start_MS[L_i]) + VI_System_Time_MS + 1;
        END_IF;

        IF (L_Desired_Code = 1) AND L_State.Confirmed_Open THEN
            L_State.Feedback_Timeout := FALSE;
        ELSIF (L_Desired_Code = 2) AND L_State.Confirmed_Closed THEN
            L_State.Feedback_Timeout := FALSE;
        ELSIF L_Elapsed_MS >= 10000 THEN
            L_State.Feedback_Timeout := TRUE;
            L_State.Travel_Timeout_Active := TRUE;
            L_State.Valve_Stuck_Suspected := TRUE;
            L_State.Valve_Degraded := TRUE;
        END_IF;
    END_IF;

    IF L_State.Feedback_Conflict THEN
        L_State.Status_Code := 3;
        L_State.Status_Text := 'Valve feedback conflict detected';
    ELSIF L_State.Feedback_Timeout THEN
        L_State.Status_Code := 2;
        L_State.Status_Text := 'Valve feedback timeout';
    ELSIF L_State.Confirmation_Unknown THEN
        L_State.Status_Code := 1;
        L_State.Status_Text := 'Valve position unknown';
    ELSE
        L_State.Status_Code := 0;
        L_State.Status_Text := 'Valve feedback healthy';
    END_IF;

    GVL_Water_Valve_Feedback.G_Valve_Feedback_State[L_i] := L_State;

    L_Any_Degraded := L_Any_Degraded OR L_State.Valve_Degraded;
    L_Any_Timeout := L_Any_Timeout OR L_State.Feedback_Timeout;
    L_Any_Conflict := L_Any_Conflict OR L_State.Feedback_Conflict;
END_FOR;

GVL_Water_Valve_Feedback.G_Any_Degraded := L_Any_Degraded;
GVL_Water_Valve_Feedback.G_Any_Timeout := L_Any_Timeout;
GVL_Water_Valve_Feedback.G_Any_Conflict := L_Any_Conflict;
GVL_Water_Valve_Feedback.G_Runtime_Valid := TRUE;
GVL_Water_Valve_Feedback.G_Last_Update_MS := VI_System_Time_MS;

IF L_Any_Conflict THEN
    GVL_Water_Valve_Feedback.G_Status_Code := 3;
    GVL_Water_Valve_Feedback.G_Status_Text := 'Valve feedback conflicts detected';
ELSIF L_Any_Timeout THEN
    GVL_Water_Valve_Feedback.G_Status_Code := 2;
    GVL_Water_Valve_Feedback.G_Status_Text := 'Valve feedback timeout detected';
ELSIF L_Any_Degraded THEN
    GVL_Water_Valve_Feedback.G_Status_Code := 1;
    GVL_Water_Valve_Feedback.G_Status_Text := 'Valve diagnostics degraded';
ELSE
    GVL_Water_Valve_Feedback.G_Status_Code := 0;
    GVL_Water_Valve_Feedback.G_Status_Text := 'Valve feedback runtime healthy';
END_IF;

END_FUNCTION_BLOCK
